KUKA KRL program: EPS_2_26115_SA7005_A_20260219035543.src

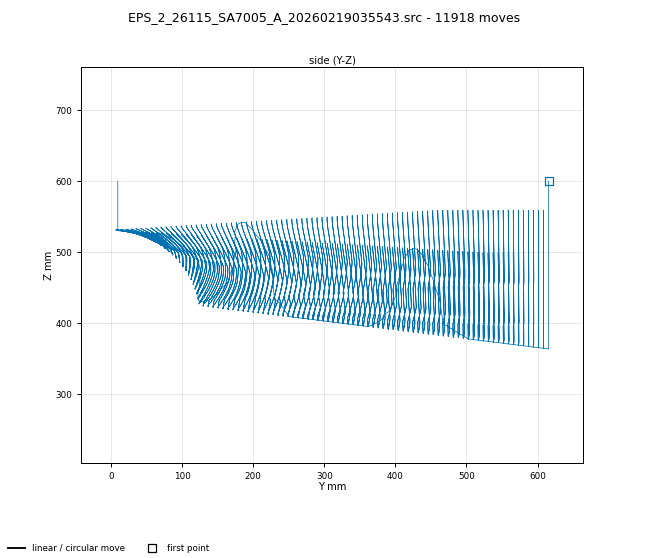
[picture p0: tool path of EPS_2_26115_SA7005_A_20260219035543.src, 11918 of 11920 moves have a stored position in this frame; points joined in program order, loops and branches not executed]
&ACCESS RVP
&REL 4
&COMMENT QRS 19112012
&PARAM EDITMASK = *
DEF PART()
EXT BAS (BAS_COMMAND :IN,REAL :IN )
INT I
BAS (#INITMOV,0 )

;KUKA QRS Post kuka4.cps  Date:22-06-2017 !

File_ID=3061

QRS_PRE_INIT()

;Init var - Until changes are made in qrs_pre_init
Outlet_Square_prg=0
Inlet_1_Square_prg=0
Inlet_2_Square_prg=0
Inlet_3_Square_prg=0
Inlet_4_Square_prg=0
Inlet_5_Square_prg=0

Outlet_1={X 0.000, Y 460.000, Z 458.500, B 0.000, E1 0.000 }
Inlet_1={X 0.000, Y 525.210, Z 398.500, B 0.000, E1 180.000 }
Outlet_1_type=201
Inlet_1_type=201
;QRS#1=Sidecore dimensions
;QRS#2=200-8" PVC SDR 35 Cut Back
;QRS#3=200-8" PVC SDR 35
;QRS#4=
;QRS#5=
;QRS#6=
;QRS#7=
;QRS#8=
;QRS#9=12-08 PSX
;QRS#10=12-08 PSX
;QRS#11=
;QRS#12=
;QRS#13=
;QRS#14=
;QRS#15=
;QRS#16=1220x127x838 2,75'
;QRS#17=EPS Height
;QRS#18=559
;QRS#19=*
;QRS#20= UPDATED VERSION 22-06-2017
;QRS#21=*
Outlet_Square=0100
Inlet_1_Square=0100
Inlet_2_Square=0
Inlet_3_Square=0
Inlet_4_Square=0
Inlet_5_Square=0
Mill_Square=1
Outlet_Square_Prg=214
Inlet_1_Square_prg=204

QRS_INIT()

$ADVANCE=5

; T1
PTP {E1 173.607,E2 173.607}
PTP {X 0,Y 615.507,A -85,B 0,C 180,E1 173.607,E2 173.607,E3 0,E4 0,E5 0,E6 0}
QRS_SPEED_INIT()
LIN {X 0,Y 615.507,Z 600,A -85,B 0,C 180,E1 173.607,E2 173.607,E3 0,E4 0,E5 0,E6 0} C_VEL
LIN {X 0,Y 615.507,Z 373.869,A -85,B 0,C 180,E1 173.607,E2 173.607} C_VEL
LIN {X 0,Y 615.507,Z 365.696,A -85,B 0,C 180,E1 173.607,E2 173.607} C_VEL
LIN {X 0,Y 615.492,Z 363.696,A -85,B 0,C 180,E1 173.421,E2 173.421} C_VEL
LIN {X 0,Y 615.49,Z 363.687,A -85,B 0,C 180,E1 170.801,E2 170.801} C_VEL
LIN {X 0,Y 615.487,Z 363.701,A -85,B 0,C 180,E1 168.139,E2 168.139} C_VEL
LIN {X 0,Y 615.481,Z 363.689,A -85,B 0,C 180,E1 165.451,E2 165.451} C_VEL
LIN {X 0,Y 615.493,Z 363.695,A -85,B 0,C 180,E1 162.73,E2 162.73} C_VEL
LIN {X 0,Y 615.49,Z 363.691,A -85,B 0,C 180,E1 159.967,E2 159.967} C_VEL
LIN {X 0,Y 615.483,Z 363.689,A -85,B 0,C 180,E1 157.155,E2 157.155} C_VEL
LIN {X 0,Y 615.486,Z 363.699,A -85,B 0,C 180,E1 154.284,E2 154.284} C_VEL
LIN {X 0,Y 615.478,Z 363.691,A -85,B 0,C 180,E1 151.552,E2 151.552} C_VEL
LIN {X 0,Y 615.487,Z 363.693,A -85,B 0,C 180,E1 148.915,E2 148.915} C_VEL
LIN {X 0,Y 615.478,Z 363.691,A -85,B 0,C 180,E1 146.468,E2 146.468} C_VEL
LIN {X 0,Y 615.493,Z 363.7,A -85,B 0,C 180,E1 144.166,E2 144.166} C_VEL
LIN {X 0,Y 615.483,Z 363.691,A -85,B 0,C 180,E1 141.931,E2 141.931} C_VEL
LIN {X 0,Y 615.482,Z 363.693,A -85,B 0,C 180,E1 139.393,E2 139.393} C_VEL
LIN {X 0,Y 615.478,Z 363.692,A -85,B 0,C 180,E1 136.754,E2 136.754} C_VEL
LIN {X 0,Y 615.491,Z 363.698,A -85,B 0,C 180,E1 133.997,E2 133.997} C_VEL
LIN {X 0,Y 615.49,Z 363.688,A -85,B 0,C 180,E1 131.474,E2 131.474} C_VEL
LIN {X 0,Y 615.49,Z 363.697,A -85,B 0,C 180,E1 128.904,E2 128.904} C_VEL
LIN {X 0,Y 615.485,Z 363.69,A -85,B 0,C 180,E1 126.425,E2 126.425} C_VEL
LIN {X 0,Y 615.485,Z 363.694,A -85,B 0,C 180,E1 125.616,E2 125.616} C_VEL
LIN {X 0,Y 615.494,Z 366.275,A -85,B 0,C 180,E1 123.236,E2 123.236} C_VEL
LIN {X 0,Y 615.479,Z 368.992,A -85,B 0,C 180,E1 120.92,E2 120.92} C_VEL
LIN {X 0,Y 615.491,Z 372.103,A -85,B 0,C 180,E1 118.45,E2 118.45} C_VEL
LIN {X 0,Y 615.498,Z 375.844,A -85,B 0,C 180,E1 115.57,E2 115.57} C_VEL
LIN {X 0,Y 615.489,Z 379.474,A -85,B 0,C 180,E1 112.845,E2 112.845} C_VEL
LIN {X 0,Y 615.479,Z 383.286,A -85,B 0,C 180,E1 110.033,E2 110.033} C_VEL
LIN {X 0,Y 615.493,Z 387.108,A -85,B 0,C 180,E1 107.27,E2 107.27} C_VEL
LIN {X 0,Y 615.482,Z 390.914,A -85,B 0,C 180,E1 104.549,E2 104.549} C_VEL
LIN {X 0,Y 615.495,Z 395.096,A -85,B 0,C 180,E1 101.61,E2 101.61} C_VEL
LIN {X 0,Y 615.494,Z 395.183,A -85,B 0,C 180,E1 101.548,E2 101.548} C_VEL
LIN {X 0,Y 615.481,Z 410.256,A -85,B 0,C 180,E1 101.193,E2 101.193} C_VEL
LIN {X 0,Y 615.494,Z 422.9,A -85,B 0,C 180,E1 100.751,E2 100.751} C_VEL
LIN {X 0,Y 615.479,Z 434.758,A -85,B 0,C 180,E1 100.195,E2 100.195} C_VEL
LIN {X 0,Y 615.499,Z 445.847,A -85,B 0,C 180,E1 99.53,E2 99.53} C_VEL
LIN {X 0,Y 615.498,Z 454.823,A -85,B 0,C 180,E1 98.867,E2 98.867} C_VEL
LIN {X 0,Y 615.498,Z 464.034,A -85,B 0,C 180,E1 98.041,E2 98.041} C_VEL
LIN {X 0,Y 615.499,Z 472.892,A -85,B 0,C 180,E1 97.057,E2 97.057} C_VEL
LIN {X 0,Y 615.497,Z 480.124,A -85,B 0,C 180,E1 96.063,E2 96.063} C_VEL
LIN {X 0,Y 615.497,Z 484.958,A -85,B 0,C 180,E1 95.241,E2 95.241} C_VEL
LIN {X 0,Y 615.494,Z 489.658,A -85,B 0,C 180,E1 94.256,E2 94.256} C_VEL
LIN {X 0,Y 615.494,Z 493.255,A -85,B 0,C 180,E1 93.273,E2 93.273} C_VEL
LIN {X 0,Y 615.496,Z 495.115,A -85,B 0,C 180,E1 92.618,E2 92.618} C_VEL
LIN {X 0,Y 615.5,Z 496.533,A -85,B 0,C 180,E1 91.963,E2 91.963} C_VEL
LIN {X 0,Y 615.496,Z 498.142,A -85,B 0,C 180,E1 90.654,E2 90.654} C_VEL
LIN {X 0,Y 615.495,Z 498.384,A -85,B 0,C 180,E1 90,E2 90} C_VEL
LIN {X 0,Y 615.495,Z 498.205,A -85,B 0,C 180,E1 89.346,E2 89.346} C_VEL
LIN {X 0,Y 615.5,Z 496.682,A -85,B 0,C 180,E1 88.037,E2 88.037} C_VEL
LIN {X 0,Y 615.498,Z 495.341,A -85,B 0,C 180,E1 87.382,E2 87.382} C_VEL
LIN {X 0,Y 615.496,Z 492.494,A -85,B 0,C 180,E1 86.399,E2 86.399} C_VEL
LIN {X 0,Y 615.498,Z 488.634,A -85,B 0,C 180,E1 85.415,E2 85.415} C_VEL
LIN {X 0,Y 615.498,Z 483.651,A -85,B 0,C 180,E1 84.43,E2 84.43} C_VEL
LIN {X 0,Y 615.496,Z 477.208,A -85,B 0,C 180,E1 83.418,E2 83.418} C_VEL
LIN {X 0,Y 615.497,Z 469.536,A -85,B 0,C 180,E1 82.454,E2 82.454} C_VEL
LIN {X 0,Y 615.498,Z 459.757,A -85,B 0,C 180,E1 81.463,E2 81.463} C_VEL
LIN {X 0,Y 615.498,Z 449.491,A -85,B 0,C 180,E1 80.636,E2 80.636} C_VEL
LIN {X 0,Y 615.482,Z 437.929,A -85,B 0,C 180,E1 79.888,E2 79.888} C_VEL
LIN {X 0,Y 615.491,Z 426.089,A -85,B 0,C 180,E1 79.294,E2 79.294} C_VEL
LIN {X 0,Y 615.477,Z 413.157,A -85,B 0,C 180,E1 78.807,E2 78.807} C_VEL
LIN {X 0,Y 615.486,Z 400.552,A -85,B 0,C 180,E1 78.473,E2 78.473} C_VEL
LIN {X 0,Y 615.494,Z 395.192,A -85,B 0,C 180,E1 78.369,E2 78.369} C_VEL
LIN {X 0,Y 615.482,Z 391.041,A -85,B 0,C 180,E1 75.451,E2 75.451} C_VEL
LIN {X 0,Y 615.497,Z 387.23,A -85,B 0,C 180,E1 72.73,E2 72.73} C_VEL
LIN {X 0,Y 615.479,Z 383.41,A -85,B 0,C 180,E1 69.967,E2 69.967} C_VEL
LIN {X 0,Y 615.492,Z 379.593,A -85,B 0,C 180,E1 67.155,E2 67.155} C_VEL
LIN {X 0,Y 615.487,Z 375.772,A -85,B 0,C 180,E1 64.284,E2 64.284} C_VEL
LIN {X 0,Y 615.492,Z 371.954,A -85,B 0,C 180,E1 61.342,E2 61.342} C_VEL
LIN {X 0,Y 615.483,Z 368.903,A -85,B 0,C 180,E1 58.915,E2 58.915} C_VEL
LIN {X 0,Y 615.495,Z 366.025,A -85,B 0,C 180,E1 56.465,E2 56.465} C_VEL
LIN {X 0,Y 615.484,Z 363.697,A -85,B 0,C 180,E1 54.384,E2 54.384} C_VEL
LIN {X 0,Y 615.481,Z 363.689,A -85,B 0,C 180,E1 51.931,E2 51.931} C_VEL
LIN {X 0,Y 615.494,Z 363.699,A -85,B 0,C 180,E1 49.394,E2 49.394} C_VEL
LIN {X 0,Y 615.496,Z 363.686,A -85,B 0,C 180,E1 46.756,E2 46.756} C_VEL
LIN {X 0,Y 615.486,Z 363.693,A -85,B 0,C 180,E1 43.997,E2 43.997} C_VEL
LIN {X 0,Y 615.488,Z 363.697,A -85,B 0,C 180,E1 41.094,E2 41.094} C_VEL
LIN {X 0,Y 615.495,Z 363.692,A -85,B 0,C 180,E1 38.904,E2 38.904} C_VEL
LIN {X 0,Y 615.478,Z 363.691,A -85,B 0,C 180,E1 36.426,E2 36.426} C_VEL
LIN {X 0,Y 615.495,Z 363.699,A -85,B 0,C 180,E1 34.022,E2 34.022} C_VEL
LIN {X 0,Y 615.482,Z 363.689,A -85,B 0,C 180,E1 31.686,E2 31.686} C_VEL
LIN {X 0,Y 615.478,Z 363.693,A -85,B 0,C 180,E1 29.407,E2 29.407} C_VEL
LIN {X 0,Y 615.498,Z 363.694,A -85,B 0,C 180,E1 27.046,E2 27.046} C_VEL
LIN {X 0,Y 615.487,Z 363.691,A -85,B 0,C 180,E1 24.272,E2 24.272} C_VEL
LIN {X 0,Y 615.479,Z 363.69,A -85,B 0,C 180,E1 21.432,E2 21.432} C_VEL
LIN {X 0,Y 615.486,Z 363.7,A -85,B 0,C 180,E1 18.603,E2 18.603} C_VEL
LIN {X 0,Y 615.477,Z 363.691,A -85,B 0,C 180,E1 15.906,E2 15.906} C_VEL
LIN {X 0,Y 615.494,Z 363.691,A -85,B 0,C 180,E1 13.201,E2 13.201} C_VEL
LIN {X 0,Y 615.486,Z 363.693,A -85,B 0,C 180,E1 10.527,E2 10.527} C_VEL
LIN {X 0,Y 615.477,Z 363.692,A -85,B 0,C 180,E1 7.876,E2 7.876} C_VEL
LIN {X 0,Y 615.496,Z 363.694,A -85,B 0,C 180,E1 5.241,E2 5.241} C_VEL
LIN {X 0,Y 615.488,Z 363.688,A -85,B 0,C 180,E1 2.618,E2 2.618} C_VEL
LIN {X 0,Y 615.487,Z 363.699,A -85,B 0,C 180,E1 0,E2 0} C_VEL
LIN {X 0,Y 615.488,Z 363.687,A -85,B 0,C 180,E1 -2.618,E2 -2.618} C_VEL
LIN {X 0,Y 615.494,Z 363.701,A -85,B 0,C 180,E1 -5.241,E2 -5.241} C_VEL
LIN {X 0,Y 615.478,Z 363.69,A -85,B 0,C 180,E1 -7.876,E2 -7.876} C_VEL
LIN {X 0,Y 615.486,Z 363.698,A -85,B 0,C 180,E1 -10.527,E2 -10.527} C_VEL
LIN {X 0,Y 615.494,Z 363.687,A -85,B 0,C 180,E1 -13.201,E2 -13.201} C_VEL
LIN {X 0,Y 615.487,Z 363.692,A -85,B 0,C 180,E1 -15.905,E2 -15.905} C_VEL
LIN {X 0,Y 615.488,Z 363.694,A -85,B 0,C 180,E1 -18.646,E2 -18.646} C_VEL
LIN {X 0,Y 615.478,Z 363.69,A -85,B 0,C 180,E1 -21.432,E2 -21.432} C_VEL
LIN {X 0,Y 615.484,Z 363.697,A -85,B 0,C 180,E1 -24.272,E2 -24.272} C_VEL
LIN {X 0,Y 615.497,Z 363.689,A -85,B 0,C 180,E1 -27.046,E2 -27.046} C_VEL
LIN {X 0,Y 615.488,Z 363.689,A -85,B 0,C 180,E1 -29.794,E2 -29.794} C_VEL
LIN {X 0,Y 615.491,Z 363.697,A -85,B 0,C 180,E1 -32.457,E2 -32.457} C_VEL
LIN {X 0,Y 615.49,Z 363.69,A -85,B 0,C 180,E1 -34.815,E2 -34.815} C_VEL
LIN {X 0,Y 615.481,Z 363.692,A -85,B 0,C 180,E1 -37.243,E2 -37.243} C_VEL
LIN {X 0,Y 615.483,Z 363.689,A -85,B 0,C 180,E1 -40.088,E2 -40.088} C_VEL
LIN {X 0,Y 615.477,Z 363.692,A -85,B 0,C 180,E1 -42.354,E2 -42.354} C_VEL
LIN {X 0,Y 615.48,Z 363.692,A -85,B 0,C 180,E1 -45.069,E2 -45.069} C_VEL
LIN {X 0,Y 615.495,Z 363.698,A -85,B 0,C 180,E1 -47.919,E2 -47.919} C_VEL
LIN {X 0,Y 615.477,Z 363.692,A -85,B 0,C 180,E1 -50.249,E2 -50.249} C_VEL
LIN {X 0,Y 615.483,Z 363.702,A -85,B 0,C 180,E1 -53.064,E2 -53.064} C_VEL
LIN {X 0,Y 615.49,Z 363.816,A -85,B 0,C 180,E1 -54.535,E2 -54.535} C_VEL
LIN {X 0,Y 615.482,Z 372.577,A -85,B 0,C 180,E1 -57.153,E2 -57.153} C_VEL
LIN {X 0,Y 615.484,Z 381.83,A -85,B 0,C 180,E1 -59.839,E2 -59.839} C_VEL
LIN {X 0,Y 615.495,Z 391.073,A -85,B 0,C 180,E1 -62.455,E2 -62.455} C_VEL
LIN {X 0,Y 615.478,Z 400.321,A -85,B 0,C 180,E1 -65.008,E2 -65.008} C_VEL
LIN {X 0,Y 615.479,Z 410.869,A -85,B 0,C 180,E1 -67.863,E2 -67.863} C_VEL
LIN {X 0,Y 615.48,Z 421.423,A -85,B 0,C 180,E1 -70.662,E2 -70.662} C_VEL
LIN {X 0,Y 615.489,Z 431.956,A -85,B 0,C 180,E1 -73.413,E2 -73.413} C_VEL
LIN {X 0,Y 615.492,Z 442.498,A -85,B 0,C 180,E1 -76.126,E2 -76.126} C_VEL
LIN {X 0,Y 615.491,Z 451.209,A -85,B 0,C 180,E1 -78.348,E2 -78.348} C_VEL
LIN {X 0,Y 615.499,Z 465.815,A -85,B 0,C 180,E1 -78.64,E2 -78.64} C_VEL
LIN {X 0,Y 615.489,Z 478.534,A -85,B 0,C 180,E1 -79.036,E2 -79.036} C_VEL
LIN {X 0,Y 615.479,Z 490.764,A -85,B 0,C 180,E1 -79.556,E2 -79.556} C_VEL
LIN {X 0,Y 615.498,Z 501.384,A -85,B 0,C 180,E1 -80.138,E2 -80.138} C_VEL
LIN {X 0,Y 615.498,Z 512.23,A -85,B 0,C 180,E1 -80.884,E2 -80.884} C_VEL
LIN {X 0,Y 615.497,Z 522.81,A -85,B 0,C 180,E1 -81.794,E2 -81.794} C_VEL
LIN {X 0,Y 615.498,Z 530.605,A -85,B 0,C 180,E1 -82.619,E2 -82.619} C_VEL
LIN {X 0,Y 615.496,Z 538.202,A -85,B 0,C 180,E1 -83.608,E2 -83.608} C_VEL
LIN {X 0,Y 615.498,Z 545.204,A -85,B 0,C 180,E1 -84.759,E2 -84.759} C_VEL
LIN {X 0,Y 615.493,Z 549.851,A -85,B 0,C 180,E1 -85.743,E2 -85.743} C_VEL
LIN {X 0,Y 615.495,Z 553.398,A -85,B 0,C 180,E1 -86.727,E2 -86.727} C_VEL
LIN {X 0,Y 615.497,Z 555.233,A -85,B 0,C 180,E1 -87.382,E2 -87.382} C_VEL
LIN {X 0,Y 615.499,Z 556.607,A -85,B 0,C 180,E1 -88.037,E2 -88.037} C_VEL
LIN {X 0,Y 615.496,Z 558.173,A -85,B 0,C 180,E1 -89.346,E2 -89.346} C_VEL
LIN {X 0,Y 615.494,Z 558.389,A -85,B 0,C 180,E1 -90,E2 -90} C_VEL
LIN {X 0,Y 615.496,Z 557.58,A -85,B 0,C 180,E1 -91.309,E2 -91.309} C_VEL
LIN {X 0,Y 615.499,Z 556.608,A -85,B 0,C 180,E1 -91.963,E2 -91.963} C_VEL
LIN {X 0,Y 615.497,Z 555.233,A -85,B 0,C 180,E1 -92.618,E2 -92.618} C_VEL
LIN {X 0,Y 615.496,Z 552.35,A -85,B 0,C 180,E1 -93.601,E2 -93.601} C_VEL
LIN {X 0,Y 615.498,Z 548.442,A -85,B 0,C 180,E1 -94.584,E2 -94.584} C_VEL
LIN {X 0,Y 615.499,Z 543.405,A -85,B 0,C 180,E1 -95.57,E2 -95.57} C_VEL
LIN {X 0,Y 615.497,Z 536.869,A -85,B 0,C 180,E1 -96.583,E2 -96.583} C_VEL
LIN {X 0,Y 615.497,Z 529.133,A -85,B 0,C 180,E1 -97.545,E2 -97.545} C_VEL
LIN {X 0,Y 615.498,Z 521.045,A -85,B 0,C 180,E1 -98.371,E2 -98.371} C_VEL
LIN {X 0,Y 615.499,Z 511.167,A -85,B 0,C 180,E1 -99.199,E2 -99.199} C_VEL
LIN {X 0,Y 615.491,Z 499.981,A -85,B 0,C 180,E1 -99.945,E2 -99.945} C_VEL
LIN {X 0,Y 615.481,Z 489.023,A -85,B 0,C 180,E1 -100.527,E2 -100.527} C_VEL
LIN {X 0,Y 615.489,Z 476.47,A -85,B 0,C 180,E1 -101.041,E2 -101.041} C_VEL
LIN {X 0,Y 615.498,Z 464.062,A -85,B 0,C 180,E1 -101.401,E2 -101.401} C_VEL
LIN {X 0,Y 615.491,Z 451.209,A -85,B 0,C 180,E1 -101.652,E2 -101.652} C_VEL
LIN {X 0,Y 615.476,Z 441.069,A -85,B 0,C 180,E1 -104.24,E2 -104.24} C_VEL
LIN {X 0,Y 615.484,Z 430.64,A -85,B 0,C 180,E1 -106.928,E2 -106.928} C_VEL
LIN {X 0,Y 615.485,Z 420.104,A -85,B 0,C 180,E1 -109.685,E2 -109.685} C_VEL
LIN {X 0,Y 615.492,Z 410.085,A -85,B 0,C 180,E1 -112.346,E2 -112.346} C_VEL
LIN {X 0,Y 615.481,Z 399.262,A -85,B 0,C 180,E1 -115.281,E2 -115.281} C_VEL
LIN {X 0,Y 615.487,Z 389.754,A -85,B 0,C 180,E1 -117.915,E2 -117.915} C_VEL
LIN {X 0,Y 615.496,Z 380.509,A -85,B 0,C 180,E1 -120.539,E2 -120.539} C_VEL
LIN {X 0,Y 615.491,Z 371.255,A -85,B 0,C 180,E1 -123.236,E2 -123.236} C_VEL
LIN {X 0,Y 615.489,Z 363.692,A -85,B 0,C 180,E1 -125.515,E2 -125.515} C_VEL
LIN {X 0,Y 615.481,Z 363.691,A -85,B 0,C 180,E1 -128.069,E2 -128.069} C_VEL
LIN {X 0,Y 615.482,Z 363.695,A -85,B 0,C 180,E1 -130.607,E2 -130.607} C_VEL
LIN {X 0,Y 615.496,Z 363.689,A -85,B 0,C 180,E1 -133.244,E2 -133.244} C_VEL
LIN {X 0,Y 615.488,Z 363.689,A -85,B 0,C 180,E1 -136.003,E2 -136.003} C_VEL
LIN {X 0,Y 615.489,Z 363.701,A -85,B 0,C 180,E1 -138.906,E2 -138.906} C_VEL
LIN {X 0,Y 615.49,Z 363.689,A -85,B 0,C 180,E1 -141.096,E2 -141.096} C_VEL
LIN {X 0,Y 615.478,Z 363.694,A -85,B 0,C 180,E1 -143.574,E2 -143.574} C_VEL
LIN {X 0,Y 615.494,Z 363.693,A -85,B 0,C 180,E1 -145.978,E2 -145.978} C_VEL
LIN {X 0,Y 615.482,Z 363.689,A -85,B 0,C 180,E1 -148.314,E2 -148.314} C_VEL
LIN {X 0,Y 615.481,Z 363.697,A -85,B 0,C 180,E1 -150.593,E2 -150.593} C_VEL
LIN {X 0,Y 615.497,Z 363.69,A -85,B 0,C 180,E1 -152.954,E2 -152.954} C_VEL
LIN {X 0,Y 615.484,Z 363.696,A -85,B 0,C 180,E1 -155.728,E2 -155.728} C_VEL
LIN {X 0,Y 615.478,Z 363.69,A -85,B 0,C 180,E1 -158.568,E2 -158.568} C_VEL
LIN {X 0,Y 615.489,Z 363.694,A -85,B 0,C 180,E1 -161.396,E2 -161.396} C_VEL
LIN {X 0,Y 615.486,Z 363.692,A -85,B 0,C 180,E1 -164.095,E2 -164.095} C_VEL
LIN {X 0,Y 615.494,Z 363.688,A -85,B 0,C 180,E1 -166.799,E2 -166.799} C_VEL
LIN {X 0,Y 615.486,Z 363.697,A -85,B 0,C 180,E1 -169.473,E2 -169.473} C_VEL
LIN {X 0,Y 615.478,Z 363.69,A -85,B 0,C 180,E1 -172.124,E2 -172.124} C_VEL
LIN {X 0,Y 615.491,Z 363.701,A -85,B 0,C 180,E1 -174.759,E2 -174.759} C_VEL
LIN {X 0,Y 615.488,Z 363.687,A -85,B 0,C 180,E1 -177.382,E2 -177.382} C_VEL
LIN {X 0,Y 615.486,Z 363.701,A -85,B 0,C 180,E1 -180,E2 -180} C_VEL
LIN {X 0,Y 615.488,Z 363.688,A -85,B 0,C 180,E1 -182.618,E2 -182.618} C_VEL
LIN {X 0,Y 615.495,Z 363.695,A -85,B 0,C 180,E1 -185.241,E2 -185.241} C_VEL
LIN {X 0,Y 615.492,Z 363.696,A -85,B 0,C 180,E1 -186.579,E2 -186.579} C_VEL
LIN {X 0,Y 614.816,Z 363.838,A -85,B 0,C 180,E1 -187.125,E2 -187.125} C_VEL
LIN {X 0,Y 611.982,Z 364.252,A -85,B 0,C 180,E1 -188.011,E2 -188.011} C_VEL
LIN {X 0,Y 609.59,Z 364.56,A -85,B 0,C 180,E1 -188.723,E2 -188.723} C_VEL
LIN {X 0,Y 608.552,Z 364.679,A -85,B 0,C 180,E1 -189.273,E2 -189.273} C_VEL
LIN {X 0,Y 608.462,Z 364.689,A -85,B 0,C 180,E1 -189.459,E2 -189.459} C_VEL
LIN {X 0,Y 608.463,Z 364.696,A -85,B 0,C 180,E1 -192,E2 -192} C_VEL
LIN {X 0,Y 608.473,Z 364.688,A -85,B 0,C 180,E1 -194.721,E2 -194.721} C_VEL
LIN {X 0,Y 608.455,Z 364.692,A -85,B 0,C 180,E1 -197.477,E2 -197.477} C_VEL
LIN {X 0,Y 608.469,Z 364.693,A -85,B 0,C 180,E1 -200.274,E2 -200.274} C_VEL
LIN {X 0,Y 608.449,Z 364.69,A -85,B 0,C 180,E1 -203.124,E2 -203.124} C_VEL
LIN {X 0,Y 608.475,Z 364.693,A -85,B 0,C 180,E1 -205.721,E2 -205.721} C_VEL
LIN {X 0,Y 608.446,Z 364.691,A -85,B 0,C 180,E1 -208.267,E2 -208.267} C_VEL
LIN {X 0,Y 608.476,Z 364.692,A -85,B 0,C 180,E1 -210.545,E2 -210.545} C_VEL
LIN {X 0,Y 608.459,Z 364.691,A -85,B 0,C 180,E1 -212.88,E2 -212.88} C_VEL
LIN {X 0,Y 608.443,Z 364.692,A -85,B 0,C 180,E1 -215.278,E2 -215.278} C_VEL
LIN {X 0,Y 608.469,Z 364.693,A -85,B 0,C 180,E1 -217.746,E2 -217.746} C_VEL
LIN {X 0,Y 608.448,Z 364.691,A -85,B 0,C 180,E1 -220.328,E2 -220.328} C_VEL
LIN {X 0,Y 608.449,Z 364.695,A -85,B 0,C 180,E1 -222.96,E2 -222.96} C_VEL
LIN {X 0,Y 608.461,Z 364.691,A -85,B 0,C 180,E1 -225.736,E2 -225.736} C_VEL
LIN {X 0,Y 608.465,Z 364.689,A -85,B 0,C 180,E1 -228.658,E2 -228.658} C_VEL
LIN {X 0,Y 608.465,Z 364.69,A -85,B 0,C 180,E1 -231.76,E2 -231.76} C_VEL
LIN {X 0,Y 608.447,Z 364.691,A -85,B 0,C 180,E1 -233.955,E2 -233.955} C_VEL
LIN {X 0,Y 608.413,Z 364.753,A -85,B 0,C 180,E1 -234.72,E2 -234.72} C_VEL
LIN {X 0,Y 608.433,Z 367.539,A -85,B 0,C 180,E1 -237.119,E2 -237.119} C_VEL
LIN {X 0,Y 608.426,Z 370.257,A -85,B 0,C 180,E1 -239.453,E2 -239.453} C_VEL
LIN {X 0,Y 608.433,Z 373.117,A -85,B 0,C 180,E1 -241.732,E2 -241.732} C_VEL
LIN {X 0,Y 608.438,Z 376.96,A -85,B 0,C 180,E1 -244.698,E2 -244.698} C_VEL
LIN {X 0,Y 608.436,Z 380.803,A -85,B 0,C 180,E1 -247.593,E2 -247.593} C_VEL
LIN {X 0,Y 608.414,Z 384.646,A -85,B 0,C 180,E1 -250.428,E2 -250.428} C_VEL
LIN {X 0,Y 608.42,Z 388.49,A -85,B 0,C 180,E1 -253.215,E2 -253.215} C_VEL
LIN {X 0,Y 608.442,Z 392.379,A -85,B 0,C 180,E1 -255.994,E2 -255.994} C_VEL
LIN {X 0,Y 608.444,Z 395.666,A -85,B 0,C 180,E1 -258.317,E2 -258.317} C_VEL
LIN {X 0,Y 608.531,Z 411.501,A -85,B 0,C 180,E1 -258.71,E2 -258.71} C_VEL
LIN {X 0,Y 608.516,Z 423.818,A -85,B 0,C 180,E1 -259.157,E2 -259.157} C_VEL
LIN {X 0,Y 608.48,Z 434.934,A -85,B 0,C 180,E1 -259.687,E2 -259.687} C_VEL
LIN {X 0,Y 608.5,Z 446.067,A -85,B 0,C 180,E1 -260.359,E2 -260.359} C_VEL
LIN {X 0,Y 608.474,Z 455.084,A -85,B 0,C 180,E1 -261.029,E2 -261.029} C_VEL
LIN {X 0,Y 608.464,Z 464.35,A -85,B 0,C 180,E1 -261.866,E2 -261.866} C_VEL
LIN {X 0,Y 608.466,Z 473.323,A -85,B 0,C 180,E1 -262.867,E2 -262.867} C_VEL
LIN {X 0,Y 608.444,Z 480.555,A -85,B 0,C 180,E1 -263.867,E2 -263.867} C_VEL
LIN {X 0,Y 608.462,Z 485.434,A -85,B 0,C 180,E1 -264.698,E2 -264.698} C_VEL
LIN {X 0,Y 608.439,Z 490.178,A -85,B 0,C 180,E1 -265.694,E2 -265.694} C_VEL
LIN {X 0,Y 608.425,Z 493.812,A -85,B 0,C 180,E1 -266.689,E2 -266.689} C_VEL
LIN {X 0,Y 608.425,Z 495.691,A -85,B 0,C 180,E1 -267.352,E2 -267.352} C_VEL
LIN {X 0,Y 608.444,Z 497.127,A -85,B 0,C 180,E1 -268.014,E2 -268.014} C_VEL
LIN {X 0,Y 608.439,Z 498.752,A -85,B 0,C 180,E1 -269.338,E2 -269.338} C_VEL
LIN {X 0,Y 608.435,Z 498.995,A -85,B 0,C 180,E1 -270,E2 -270} C_VEL
LIN {X 0,Y 608.438,Z 498.815,A -85,B 0,C 180,E1 -270.662,E2 -270.662} C_VEL
LIN {X 0,Y 608.445,Z 497.276,A -85,B 0,C 180,E1 -271.986,E2 -271.986} C_VEL
LIN {X 0,Y 608.426,Z 495.918,A -85,B 0,C 180,E1 -272.648,E2 -272.648} C_VEL
LIN {X 0,Y 608.449,Z 493.041,A -85,B 0,C 180,E1 -273.642,E2 -273.642} C_VEL
LIN {X 0,Y 608.433,Z 489.142,A -85,B 0,C 180,E1 -274.638,E2 -274.638} C_VEL
LIN {X 0,Y 608.45,Z 484.111,A -85,B 0,C 180,E1 -275.635,E2 -275.635} C_VEL
LIN {X 0,Y 608.441,Z 477.794,A -85,B 0,C 180,E1 -276.633,E2 -276.633} C_VEL
LIN {X 0,Y 608.475,Z 469.877,A -85,B 0,C 180,E1 -277.633,E2 -277.633} C_VEL
LIN {X 0,Y 608.472,Z 460.035,A -85,B 0,C 180,E1 -278.636,E2 -278.636} C_VEL
LIN {X 0,Y 608.481,Z 449.712,A -85,B 0,C 180,E1 -279.473,E2 -279.473} C_VEL
LIN {X 0,Y 608.478,Z 438.097,A -85,B 0,C 180,E1 -280.229,E2 -280.229} C_VEL
LIN {X 0,Y 608.507,Z 426.22,A -85,B 0,C 180,E1 -280.831,E2 -280.831} C_VEL
LIN {X 0,Y 608.521,Z 413.257,A -85,B 0,C 180,E1 -281.323,E2 -281.323} C_VEL
LIN {X 0,Y 608.546,Z 400.638,A -85,B 0,C 180,E1 -281.66,E2 -281.66} C_VEL
LIN {X 0,Y 608.441,Z 395.674,A -85,B 0,C 180,E1 -281.768,E2 -281.768} C_VEL
LIN {X 0,Y 608.423,Z 392.46,A -85,B 0,C 180,E1 -284.039,E2 -284.039} C_VEL
LIN {X 0,Y 608.421,Z 388.615,A -85,B 0,C 180,E1 -286.785,E2 -286.785} C_VEL
LIN {X 0,Y 608.416,Z 384.769,A -85,B 0,C 180,E1 -289.572,E2 -289.572} C_VEL
LIN {X 0,Y 608.433,Z 380.84,A -85,B 0,C 180,E1 -292.469,E2 -292.469} C_VEL
LIN {X 0,Y 608.438,Z 377.078,A -85,B 0,C 180,E1 -295.302,E2 -295.302} C_VEL
LIN {X 0,Y 608.433,Z 373.232,A -85,B 0,C 180,E1 -298.268,E2 -298.268} C_VEL
LIN {X 0,Y 608.429,Z 370.361,A -85,B 0,C 180,E1 -300.547,E2 -300.547} C_VEL
LIN {X 0,Y 608.434,Z 367.65,A -85,B 0,C 180,E1 -302.881,E2 -302.881} C_VEL
LIN {X 0,Y 608.44,Z 364.856,A -85,B 0,C 180,E1 -305.278,E2 -305.278} C_VEL
LIN {X 0,Y 608.469,Z 364.689,A -85,B 0,C 180,E1 -307.747,E2 -307.747} C_VEL
LIN {X 0,Y 608.453,Z 364.695,A -85,B 0,C 180,E1 -310.329,E2 -310.329} C_VEL
LIN {X 0,Y 608.483,Z 364.687,A -85,B 0,C 180,E1 -313.31,E2 -313.31} C_VEL
LIN {X 0,Y 608.47,Z 364.69,A -85,B 0,C 180,E1 -316.13,E2 -316.13} C_VEL
LIN {X 0,Y 608.456,Z 364.694,A -85,B 0,C 180,E1 -318.823,E2 -318.823} C_VEL
LIN {X 0,Y 608.474,Z 364.688,A -85,B 0,C 180,E1 -321.412,E2 -321.412} C_VEL
LIN {X 0,Y 608.453,Z 364.694,A -85,B 0,C 180,E1 -323.954,E2 -323.954} C_VEL
LIN {X 0,Y 608.45,Z 364.693,A -85,B 0,C 180,E1 -326.328,E2 -326.328} C_VEL
LIN {X 0,Y 608.45,Z 364.691,A -85,B 0,C 180,E1 -328.733,E2 -328.733} C_VEL
LIN {X 0,Y 608.468,Z 364.691,A -85,B 0,C 180,E1 -331.382,E2 -331.382} C_VEL
LIN {X 0,Y 608.438,Z 364.693,A -85,B 0,C 180,E1 -333.964,E2 -333.964} C_VEL
LIN {X 0,Y 608.473,Z 364.696,A -85,B 0,C 180,E1 -336.155,E2 -336.155} C_VEL
LIN {X 0,Y 608.456,Z 364.69,A -85,B 0,C 180,E1 -339.018,E2 -339.018} C_VEL
LIN {X 0,Y 608.447,Z 364.692,A -85,B 0,C 180,E1 -341.828,E2 -341.828} C_VEL
LIN {X 0,Y 608.471,Z 364.694,A -85,B 0,C 180,E1 -344.594,E2 -344.594} C_VEL
LIN {X 0,Y 608.476,Z 364.687,A -85,B 0,C 180,E1 -347.323,E2 -347.323} C_VEL
LIN {X 0,Y 608.456,Z 364.695,A -85,B 0,C 180,E1 -350.023,E2 -350.023} C_VEL
LIN {X 0,Y 608.466,Z 364.689,A -85,B 0,C 180,E1 -352.701,E2 -352.701} C_VEL
LIN {X 0,Y 608.457,Z 364.692,A -85,B 0,C 180,E1 -355.362,E2 -355.362} C_VEL
LIN {X 0,Y 608.45,Z 364.693,A -85,B 0,C 180,E1 -358.014,E2 -358.014} C_VEL
LIN {X 0,Y 608.479,Z 364.688,A -85,B 0,C 180,E1 -360.662,E2 -360.662} C_VEL
LIN {X 0,Y 608.478,Z 364.691,A -85,B 0,C 180,E1 -363.311,E2 -363.311} C_VEL
LIN {X 0,Y 608.454,Z 364.69,A -85,B 0,C 180,E1 -365.967,E2 -365.967} C_VEL
LIN {X 0,Y 608.465,Z 364.696,A -85,B 0,C 180,E1 -368.636,E2 -368.636} C_VEL
LIN {X 0,Y 608.478,Z 364.687,A -85,B 0,C 180,E1 -371.324,E2 -371.324} C_VEL
LIN {X 0,Y 608.476,Z 364.692,A -85,B 0,C 180,E1 -374.037,E2 -374.037} C_VEL
LIN {X 0,Y 608.445,Z 364.693,A -85,B 0,C 180,E1 -376.784,E2 -376.784} C_VEL
LIN {X 0,Y 608.455,Z 364.69,A -85,B 0,C 180,E1 -379.571,E2 -379.571} C_VEL
LIN {X 0,Y 608.464,Z 364.695,A -85,B 0,C 180,E1 -382.476,E2 -382.476} C_VEL
LIN {X 0,Y 608.456,Z 364.691,A -85,B 0,C 180,E1 -384.571,E2 -384.571} C_VEL
LIN {X 0,Y 608.487,Z 364.69,A -85,B 0,C 180,E1 -387.208,E2 -387.208} C_VEL
LIN {X 0,Y 608.47,Z 364.688,A -85,B 0,C 180,E1 -389.971,E2 -389.971} C_VEL
LIN {X 0,Y 608.458,Z 364.693,A -85,B 0,C 180,E1 -392.88,E2 -392.88} C_VEL
LIN {X 0,Y 608.442,Z 364.692,A -85,B 0,C 180,E1 -395.278,E2 -395.278} C_VEL
LIN {X 0,Y 608.467,Z 364.696,A -85,B 0,C 180,E1 -397.747,E2 -397.747} C_VEL
LIN {X 0,Y 608.447,Z 364.691,A -85,B 0,C 180,E1 -400.328,E2 -400.328} C_VEL
LIN {X 0,Y 608.454,Z 364.697,A -85,B 0,C 180,E1 -402.96,E2 -402.96} C_VEL
LIN {X 0,Y 608.463,Z 364.69,A -85,B 0,C 180,E1 -405.736,E2 -405.736} C_VEL
LIN {X 0,Y 608.464,Z 364.689,A -85,B 0,C 180,E1 -408.658,E2 -408.658} C_VEL
LIN {X 0,Y 608.464,Z 364.692,A -85,B 0,C 180,E1 -411.76,E2 -411.76} C_VEL
LIN {X 0,Y 608.482,Z 364.814,A -85,B 0,C 180,E1 -414.369,E2 -414.369} C_VEL
LIN {X 0,Y 608.528,Z 372.592,A -85,B 0,C 180,E1 -416.73,E2 -416.73} C_VEL
LIN {X 0,Y 608.536,Z 381.859,A -85,B 0,C 180,E1 -419.459,E2 -419.459} C_VEL
LIN {X 0,Y 608.509,Z 392.45,A -85,B 0,C 180,E1 -422.485,E2 -422.485} C_VEL
LIN {X 0,Y 608.469,Z 401.718,A -85,B 0,C 180,E1 -425.065,E2 -425.065} C_VEL
LIN {X 0,Y 608.479,Z 412.309,A -85,B 0,C 180,E1 -427.952,E2 -427.952} C_VEL
LIN {X 0,Y 608.453,Z 422.9,A -85,B 0,C 180,E1 -430.78,E2 -430.78} C_VEL
LIN {X 0,Y 608.442,Z 433.181,A -85,B 0,C 180,E1 -433.48,E2 -433.48} C_VEL
LIN {X 0,Y 608.446,Z 444.146,A -85,B 0,C 180,E1 -436.319,E2 -436.319} C_VEL
LIN {X 0,Y 608.442,Z 451.53,A -85,B 0,C 180,E1 -438.211,E2 -438.211} C_VEL
LIN {X 0,Y 608.544,Z 466.691,A -85,B 0,C 180,E1 -438.53,E2 -438.53} C_VEL
LIN {X 0,Y 608.526,Z 478.239,A -85,B 0,C 180,E1 -438.893,E2 -438.893} C_VEL
LIN {X 0,Y 608.51,Z 490.918,A -85,B 0,C 180,E1 -439.435,E2 -439.435} C_VEL
LIN {X 0,Y 608.489,Z 501.576,A -85,B 0,C 180,E1 -440.023,E2 -440.023} C_VEL
LIN {X 0,Y 608.483,Z 512.472,A -85,B 0,C 180,E1 -440.778,E2 -440.778} C_VEL
LIN {X 0,Y 608.475,Z 523.11,A -85,B 0,C 180,E1 -441.699,E2 -441.699} C_VEL
LIN {X 0,Y 608.471,Z 530.959,A -85,B 0,C 180,E1 -442.534,E2 -442.534} C_VEL
LIN {X 0,Y 608.461,Z 538.286,A -85,B 0,C 180,E1 -443.484,E2 -443.484} C_VEL
LIN {X 0,Y 608.45,Z 543.865,A -85,B 0,C 180,E1 -444.365,E2 -444.365} C_VEL
LIN {X 0,Y 608.432,Z 548.95,A -85,B 0,C 180,E1 -445.362,E2 -445.362} C_VEL
LIN {X 0,Y 608.449,Z 552.896,A -85,B 0,C 180,E1 -446.358,E2 -446.358} C_VEL
LIN {X 0,Y 608.425,Z 555.809,A -85,B 0,C 180,E1 -447.352,E2 -447.352} C_VEL
LIN {X 0,Y 608.444,Z 557.201,A -85,B 0,C 180,E1 -448.014,E2 -448.014} C_VEL
LIN {X 0,Y 608.438,Z 558.783,A -85,B 0,C 180,E1 -449.338,E2 -449.338} C_VEL
LIN {X 0,Y 608.434,Z 559,A -85,B 0,C 180,E1 -450,E2 -450} C_VEL
LIN {X 0,Y 608.448,Z 558.184,A -85,B 0,C 180,E1 -451.324,E2 -451.324} C_VEL
LIN {X 0,Y 608.444,Z 557.201,A -85,B 0,C 180,E1 -451.986,E2 -451.986} C_VEL
LIN {X 0,Y 608.425,Z 555.809,A -85,B 0,C 180,E1 -452.648,E2 -452.648} C_VEL
LIN {X 0,Y 608.449,Z 552.896,A -85,B 0,C 180,E1 -453.642,E2 -453.642} C_VEL
LIN {X 0,Y 608.432,Z 548.95,A -85,B 0,C 180,E1 -454.638,E2 -454.638} C_VEL
LIN {X 0,Y 608.437,Z 542.877,A -85,B 0,C 180,E1 -455.801,E2 -455.801} C_VEL
LIN {X 0,Y 608.462,Z 536.235,A -85,B 0,C 180,E1 -456.799,E2 -456.799} C_VEL
LIN {X 0,Y 608.456,Z 527.989,A -85,B 0,C 180,E1 -457.8,E2 -457.8} C_VEL
LIN {X 0,Y 608.472,Z 519.536,A -85,B 0,C 180,E1 -458.636,E2 -458.636} C_VEL
LIN {X 0,Y 608.481,Z 509.09,A -85,B 0,C 180,E1 -459.473,E2 -459.473} C_VEL
LIN {X 0,Y 608.491,Z 498.755,A -85,B 0,C 180,E1 -460.145,E2 -460.145} C_VEL
LIN {X 0,Y 608.518,Z 487.259,A -85,B 0,C 180,E1 -460.74,E2 -460.74} C_VEL
LIN {X 0,Y 608.537,Z 474.891,A -85,B 0,C 180,E1 -461.225,E2 -461.225} C_VEL
LIN {X 0,Y 608.546,Z 461.438,A -85,B 0,C 180,E1 -461.597,E2 -461.597} C_VEL
LIN {X 0,Y 608.442,Z 451.53,A -85,B 0,C 180,E1 -461.789,E2 -461.789} C_VEL
LIN {X 0,Y 608.442,Z 441.435,A -85,B 0,C 180,E1 -464.379,E2 -464.379} C_VEL
LIN {X 0,Y 608.442,Z 430.844,A -85,B 0,C 180,E1 -467.13,E2 -467.13} C_VEL
LIN {X 0,Y 608.458,Z 421.577,A -85,B 0,C 180,E1 -469.57,E2 -469.57} C_VEL
LIN {X 0,Y 608.467,Z 410.72,A -85,B 0,C 180,E1 -472.477,E2 -472.477} C_VEL
LIN {X 0,Y 608.473,Z 400.394,A -85,B 0,C 180,E1 -475.3,E2 -475.3} C_VEL
LIN {X 0,Y 608.5,Z 391.127,A -85,B 0,C 180,E1 -477.889,E2 -477.889} C_VEL
LIN {X 0,Y 608.536,Z 381.859,A -85,B 0,C 180,E1 -480.541,E2 -480.541} C_VEL
LIN {X 0,Y 608.528,Z 372.592,A -85,B 0,C 180,E1 -483.27,E2 -483.27} C_VEL
LIN {X 0,Y 608.475,Z 364.691,A -85,B 0,C 180,E1 -485.682,E2 -485.682} C_VEL
LIN {X 0,Y 608.464,Z 364.692,A -85,B 0,C 180,E1 -488.24,E2 -488.24} C_VEL
LIN {X 0,Y 608.463,Z 364.689,A -85,B 0,C 180,E1 -491.342,E2 -491.342} C_VEL
LIN {X 0,Y 608.463,Z 364.69,A -85,B 0,C 180,E1 -494.264,E2 -494.264} C_VEL
LIN {X 0,Y 608.45,Z 364.697,A -85,B 0,C 180,E1 -497.04,E2 -497.04} C_VEL
LIN {X 0,Y 608.456,Z 364.69,A -85,B 0,C 180,E1 -499.697,E2 -499.697} C_VEL
LIN {X 0,Y 608.467,Z 364.696,A -85,B 0,C 180,E1 -502.253,E2 -502.253} C_VEL
LIN {X 0,Y 608.454,Z 364.691,A -85,B 0,C 180,E1 -505.094,E2 -505.094} C_VEL
LIN {X 0,Y 608.468,Z 364.69,A -85,B 0,C 180,E1 -507.906,E2 -507.906} C_VEL
LIN {X 0,Y 608.473,Z 364.688,A -85,B 0,C 180,E1 -510.221,E2 -510.221} C_VEL
LIN {X 0,Y 608.487,Z 364.69,A -85,B 0,C 180,E1 -512.792,E2 -512.792} C_VEL
LIN {X 0,Y 608.455,Z 364.691,A -85,B 0,C 180,E1 -515.429,E2 -515.429} C_VEL
LIN {X 0,Y 608.468,Z 364.689,A -85,B 0,C 180,E1 -518.308,E2 -518.308} C_VEL
LIN {X 0,Y 608.46,Z 364.697,A -85,B 0,C 180,E1 -521.13,E2 -521.13} C_VEL
LIN {X 0,Y 608.461,Z 364.69,A -85,B 0,C 180,E1 -523.906,E2 -523.906} C_VEL
LIN {X 0,Y 608.472,Z 364.69,A -85,B 0,C 180,E1 -526.644,E2 -526.644} C_VEL
LIN {X 0,Y 608.462,Z 364.692,A -85,B 0,C 180,E1 -529.35,E2 -529.35} C_VEL
LIN {X 0,Y 608.474,Z 364.688,A -85,B 0,C 180,E1 -532.033,E2 -532.033} C_VEL
LIN {X 0,Y 608.469,Z 364.695,A -85,B 0,C 180,E1 -534.698,E2 -534.698} C_VEL
LIN {X 0,Y 608.479,Z 364.687,A -85,B 0,C 180,E1 -537.352,E2 -537.352} C_VEL
LIN {X 0,Y 608.478,Z 364.694,A -85,B 0,C 180,E1 -540,E2 -540} C_VEL
LIN {X 0,Y 608.479,Z 364.687,A -85,B 0,C 180,E1 -542.648,E2 -542.648} C_VEL
LIN {X 0,Y 608.473,Z 364.692,A -85,B 0,C 180,E1 -545.302,E2 -545.302} C_VEL
LIN {X 0,Y 608.473,Z 364.689,A -85,B 0,C 180,E1 -547.967,E2 -547.967} C_VEL
LIN {X 0,Y 608.462,Z 364.689,A -85,B 0,C 180,E1 -549.459,E2 -549.459} C_VEL
LIN {X 0,Y 607.78,Z 364.781,A -85,B 0,C 180,E1 -550.012,E2 -550.012} C_VEL
LIN {X 0,Y 604.925,Z 365.135,A -85,B 0,C 180,E1 -550.908,E2 -550.908} C_VEL
LIN {X 0,Y 602.524,Z 365.435,A -85,B 0,C 180,E1 -551.63,E2 -551.63} C_VEL
LIN {X 0,Y 601.494,Z 365.561,A -85,B 0,C 180,E1 -552.187,E2 -552.187} C_VEL
LIN {X 0,Y 601.411,Z 365.569,A -85,B 0,C 180,E1 -552.375,E2 -552.375} C_VEL
LIN {X 0,Y 601.429,Z 365.567,A -85,B 0,C 180,E1 -554.897,E2 -554.897} C_VEL
LIN {X 0,Y 601.426,Z 365.573,A -85,B 0,C 180,E1 -556.986,E2 -556.986} C_VEL
LIN {X 0,Y 601.411,Z 365.568,A -85,B 0,C 180,E1 -559.809,E2 -559.809} C_VEL
LIN {X 0,Y 601.416,Z 365.568,A -85,B 0,C 180,E1 -562.683,E2 -562.683} C_VEL
LIN {X 0,Y 601.408,Z 365.568,A -85,B 0,C 180,E1 -564.878,E2 -564.878} C_VEL
LIN {X 0,Y 601.423,Z 365.573,A -85,B 0,C 180,E1 -567.363,E2 -567.363} C_VEL
LIN {X 0,Y 601.433,Z 365.566,A -85,B 0,C 180,E1 -570.164,E2 -570.164} C_VEL
LIN {X 0,Y 601.427,Z 365.569,A -85,B 0,C 180,E1 -572.716,E2 -572.716} C_VEL
LIN {X 0,Y 601.401,Z 365.569,A -85,B 0,C 180,E1 -575.112,E2 -575.112} C_VEL
LIN {X 0,Y 601.439,Z 365.569,A -85,B 0,C 180,E1 -577.419,E2 -577.419} C_VEL
LIN {X 0,Y 601.415,Z 365.567,A -85,B 0,C 180,E1 -579.995,E2 -579.995} C_VEL
LIN {X 0,Y 601.41,Z 365.575,A -85,B 0,C 180,E1 -582.671,E2 -582.671} C_VEL
LIN {X 0,Y 601.43,Z 365.565,A -85,B 0,C 180,E1 -585.482,E2 -585.482} C_VEL
LIN {X 0,Y 601.429,Z 365.566,A -85,B 0,C 180,E1 -588.407,E2 -588.407} C_VEL
LIN {X 0,Y 601.435,Z 365.569,A -85,B 0,C 180,E1 -591.529,E2 -591.529} C_VEL
LIN {X 0,Y 601.379,Z 365.573,A -85,B 0,C 180,E1 -594.245,E2 -594.245} C_VEL
LIN {X 0,Y 601.357,Z 365.822,A -85,B 0,C 180,E1 -595.064,E2 -595.064} C_VEL
LIN {X 0,Y 601.378,Z 368.588,A -85,B 0,C 180,E1 -597.481,E2 -597.481} C_VEL
LIN {X 0,Y 601.355,Z 371.32,A -85,B 0,C 180,E1 -599.864,E2 -599.864} C_VEL
LIN {X 0,Y 601.345,Z 374.743,A -85,B 0,C 180,E1 -602.651,E2 -602.651} C_VEL
LIN {X 0,Y 601.349,Z 377.922,A -85,B 0,C 180,E1 -605.119,E2 -605.119} C_VEL
LIN {X 0,Y 601.337,Z 381.765,A -85,B 0,C 180,E1 -608.038,E2 -608.038} C_VEL
LIN {X 0,Y 601.316,Z 384.647,A -85,B 0,C 180,E1 -610.187,E2 -610.187} C_VEL
LIN {X 0,Y 601.338,Z 388.49,A -85,B 0,C 180,E1 -613.011,E2 -613.011} C_VEL
LIN {X 0,Y 601.35,Z 392.534,A -85,B 0,C 180,E1 -615.937,E2 -615.937} C_VEL
LIN {X 0,Y 601.347,Z 395.667,A -85,B 0,C 180,E1 -618.177,E2 -618.177} C_VEL
LIN {X 0,Y 601.591,Z 401.34,A -85,B 0,C 180,E1 -618.31,E2 -618.31} C_VEL
LIN {X 0,Y 601.557,Z 414.026,A -85,B 0,C 180,E1 -618.66,E2 -618.66} C_VEL
LIN {X 0,Y 601.543,Z 426.615,A -85,B 0,C 180,E1 -619.15,E2 -619.15} C_VEL
LIN {X 0,Y 601.503,Z 438.007,A -85,B 0,C 180,E1 -619.736,E2 -619.736} C_VEL
LIN {X 0,Y 601.462,Z 449.637,A -85,B 0,C 180,E1 -620.5,E2 -620.5} C_VEL
LIN {X 0,Y 601.436,Z 459.023,A -85,B 0,C 180,E1 -621.262,E2 -621.262} C_VEL
LIN {X 0,Y 601.4,Z 467.59,A -85,B 0,C 180,E1 -622.108,E2 -622.108} C_VEL
LIN {X 0,Y 601.388,Z 475.906,A -85,B 0,C 180,E1 -623.12,E2 -623.12} C_VEL
LIN {X 0,Y 601.373,Z 482.607,A -85,B 0,C 180,E1 -624.131,E2 -624.131} C_VEL
LIN {X 0,Y 601.335,Z 488.754,A -85,B 0,C 180,E1 -625.307,E2 -625.307} C_VEL
LIN {X 0,Y 601.367,Z 492.743,A -85,B 0,C 180,E1 -626.315,E2 -626.315} C_VEL
LIN {X 0,Y 601.324,Z 495.693,A -85,B 0,C 180,E1 -627.32,E2 -627.32} C_VEL
LIN {X 0,Y 601.343,Z 497.127,A -85,B 0,C 180,E1 -627.991,E2 -627.991} C_VEL
LIN {X 0,Y 601.339,Z 498.753,A -85,B 0,C 180,E1 -629.33,E2 -629.33} C_VEL
LIN {X 0,Y 601.336,Z 498.996,A -85,B 0,C 180,E1 -630,E2 -630} C_VEL
LIN {X 0,Y 601.339,Z 498.815,A -85,B 0,C 180,E1 -630.67,E2 -630.67} C_VEL
LIN {X 0,Y 601.343,Z 497.275,A -85,B 0,C 180,E1 -632.009,E2 -632.009} C_VEL
LIN {X 0,Y 601.326,Z 495.916,A -85,B 0,C 180,E1 -632.68,E2 -632.68} C_VEL
LIN {X 0,Y 601.368,Z 493.04,A -85,B 0,C 180,E1 -633.685,E2 -633.685} C_VEL
LIN {X 0,Y 601.337,Z 489.14,A -85,B 0,C 180,E1 -634.693,E2 -634.693} C_VEL
LIN {X 0,Y 601.373,Z 484.109,A -85,B 0,C 180,E1 -635.701,E2 -635.701} C_VEL
LIN {X 0,Y 601.382,Z 477.79,A -85,B 0,C 180,E1 -636.711,E2 -636.711} C_VEL
LIN {X 0,Y 601.396,Z 469.873,A -85,B 0,C 180,E1 -637.724,E2 -637.724} C_VEL
LIN {X 0,Y 601.437,Z 460.028,A -85,B 0,C 180,E1 -638.738,E2 -638.738} C_VEL
LIN {X 0,Y 601.451,Z 449.706,A -85,B 0,C 180,E1 -639.585,E2 -639.585} C_VEL
LIN {X 0,Y 601.481,Z 438.087,A -85,B 0,C 180,E1 -640.349,E2 -640.349} C_VEL
LIN {X 0,Y 601.523,Z 426.209,A -85,B 0,C 180,E1 -640.958,E2 -640.958} C_VEL
LIN {X 0,Y 601.543,Z 413.241,A -85,B 0,C 180,E1 -641.456,E2 -641.456} C_VEL
LIN {X 0,Y 601.614,Z 400.615,A -85,B 0,C 180,E1 -641.796,E2 -641.796} C_VEL
LIN {X 0,Y 601.342,Z 395.673,A -85,B 0,C 180,E1 -641.909,E2 -641.909} C_VEL
LIN {X 0,Y 601.319,Z 392.459,A -85,B 0,C 180,E1 -644.208,E2 -644.208} C_VEL
LIN {X 0,Y 601.34,Z 388.614,A -85,B 0,C 180,E1 -646.989,E2 -646.989} C_VEL
LIN {X 0,Y 601.317,Z 384.768,A -85,B 0,C 180,E1 -649.813,E2 -649.813} C_VEL
LIN {X 0,Y 601.337,Z 381.055,A -85,B 0,C 180,E1 -652.587,E2 -652.587} C_VEL
LIN {X 0,Y 601.349,Z 378.039,A -85,B 0,C 180,E1 -654.881,E2 -654.881} C_VEL
LIN {X 0,Y 601.346,Z 374.858,A -85,B 0,C 180,E1 -657.349,E2 -657.349} C_VEL
LIN {X 0,Y 601.352,Z 371.368,A -85,B 0,C 180,E1 -660.169,E2 -660.169} C_VEL
LIN {X 0,Y 601.366,Z 368.513,A -85,B 0,C 180,E1 -662.707,E2 -662.707} C_VEL
LIN {X 0,Y 601.384,Z 365.723,A -85,B 0,C 180,E1 -665.11,E2 -665.11} C_VEL
LIN {X 0,Y 601.44,Z 365.567,A -85,B 0,C 180,E1 -667.419,E2 -667.419} C_VEL
LIN {X 0,Y 601.406,Z 365.569,A -85,B 0,C 180,E1 -669.996,E2 -669.996} C_VEL
LIN {X 0,Y 601.416,Z 365.569,A -85,B 0,C 180,E1 -672.67,E2 -672.67} C_VEL
LIN {X 0,Y 601.43,Z 365.566,A -85,B 0,C 180,E1 -674.535,E2 -674.535} C_VEL
LIN {X 0,Y 601.411,Z 365.575,A -85,B 0,C 180,E1 -677.41,E2 -677.41} C_VEL
LIN {X 0,Y 601.446,Z 365.566,A -85,B 0,C 180,E1 -680.464,E2 -680.464} C_VEL
LIN {X 0,Y 601.407,Z 365.568,A -85,B 0,C 180,E1 -683.417,E2 -683.417} C_VEL
LIN {X 0,Y 601.437,Z 365.57,A -85,B 0,C 180,E1 -686.064,E2 -686.064} C_VEL
LIN {X 0,Y 601.424,Z 365.566,A -85,B 0,C 180,E1 -688.546,E2 -688.546} C_VEL
LIN {X 0,Y 601.428,Z 365.568,A -85,B 0,C 180,E1 -691.373,E2 -691.373} C_VEL
LIN {X 0,Y 601.401,Z 365.569,A -85,B 0,C 180,E1 -693.636,E2 -693.636} C_VEL
LIN {X 0,Y 601.463,Z 365.564,A -85,B 0,C 180,E1 -695.86,E2 -695.86} C_VEL
LIN {X 0,Y 601.408,Z 365.568,A -85,B 0,C 180,E1 -698.761,E2 -698.761} C_VEL
LIN {X 0,Y 601.421,Z 365.57,A -85,B 0,C 180,E1 -701.608,E2 -701.608} C_VEL
LIN {X 0,Y 601.414,Z 365.57,A -85,B 0,C 180,E1 -704.409,E2 -704.409} C_VEL
LIN {X 0,Y 601.422,Z 365.566,A -85,B 0,C 180,E1 -707.172,E2 -707.172} C_VEL
LIN {X 0,Y 601.434,Z 365.572,A -85,B 0,C 180,E1 -709.905,E2 -709.905} C_VEL
LIN {X 0,Y 601.443,Z 365.564,A -85,B 0,C 180,E1 -712.615,E2 -712.615} C_VEL
LIN {X 0,Y 601.426,Z 365.569,A -85,B 0,C 180,E1 -715.308,E2 -715.308} C_VEL
LIN {X 0,Y 601.421,Z 365.568,A -85,B 0,C 180,E1 -717.991,E2 -717.991} C_VEL
LIN {X 0,Y 601.451,Z 365.563,A -85,B 0,C 180,E1 -720.669,E2 -720.669} C_VEL
LIN {X 0,Y 601.43,Z 365.57,A -85,B 0,C 180,E1 -723.35,E2 -723.35} C_VEL
LIN {X 0,Y 601.409,Z 365.568,A -85,B 0,C 180,E1 -726.037,E2 -726.037} C_VEL
LIN {X 0,Y 601.444,Z 365.57,A -85,B 0,C 180,E1 -728.738,E2 -728.738} C_VEL
LIN {X 0,Y 601.437,Z 365.565,A -85,B 0,C 180,E1 -731.458,E2 -731.458} C_VEL
LIN {X 0,Y 601.425,Z 365.568,A -85,B 0,C 180,E1 -734.205,E2 -734.205} C_VEL
LIN {X 0,Y 601.418,Z 365.571,A -85,B 0,C 180,E1 -736.986,E2 -736.986} C_VEL
LIN {X 0,Y 601.41,Z 365.568,A -85,B 0,C 180,E1 -739.809,E2 -739.809} C_VEL
LIN {X 0,Y 601.417,Z 365.57,A -85,B 0,C 180,E1 -742.683,E2 -742.683} C_VEL
LIN {X 0,Y 601.404,Z 365.568,A -85,B 0,C 180,E1 -744.879,E2 -744.879} C_VEL
LIN {X 0,Y 601.425,Z 365.572,A -85,B 0,C 180,E1 -747.363,E2 -747.363} C_VEL
LIN {X 0,Y 601.434,Z 365.565,A -85,B 0,C 180,E1 -750.164,E2 -750.164} C_VEL
LIN {X 0,Y 601.426,Z 365.572,A -85,B 0,C 180,E1 -752.715,E2 -752.715} C_VEL
LIN {X 0,Y 601.4,Z 365.569,A -85,B 0,C 180,E1 -755.112,E2 -755.112} C_VEL
LIN {X 0,Y 601.437,Z 365.567,A -85,B 0,C 180,E1 -757.419,E2 -757.419} C_VEL
LIN {X 0,Y 601.416,Z 365.568,A -85,B 0,C 180,E1 -759.995,E2 -759.995} C_VEL
LIN {X 0,Y 601.412,Z 365.572,A -85,B 0,C 180,E1 -762.67,E2 -762.67} C_VEL
LIN {X 0,Y 601.431,Z 365.565,A -85,B 0,C 180,E1 -765.482,E2 -765.482} C_VEL
LIN {X 0,Y 601.429,Z 365.568,A -85,B 0,C 180,E1 -768.407,E2 -768.407} C_VEL
LIN {X 0,Y 601.432,Z 365.572,A -85,B 0,C 180,E1 -771.529,E2 -771.529} C_VEL
LIN {X 0,Y 601.454,Z 365.684,A -85,B 0,C 180,E1 -774.16,E2 -774.16} C_VEL
LIN {X 0,Y 601.584,Z 372.843,A -85,B 0,C 180,E1 -776.371,E2 -776.371} C_VEL
LIN {X 0,Y 601.534,Z 381.859,A -85,B 0,C 180,E1 -779.064,E2 -779.064} C_VEL
LIN {X 0,Y 601.503,Z 391.126,A -85,B 0,C 180,E1 -781.757,E2 -781.757} C_VEL
LIN {X 0,Y 601.478,Z 400.394,A -85,B 0,C 180,E1 -784.384,E2 -784.384} C_VEL
LIN {X 0,Y 601.429,Z 409.661,A -85,B 0,C 180,E1 -786.954,E2 -786.954} C_VEL
LIN {X 0,Y 601.425,Z 420.252,A -85,B 0,C 180,E1 -789.835,E2 -789.835} C_VEL
LIN {X 0,Y 601.39,Z 430.844,A -85,B 0,C 180,E1 -792.662,E2 -792.662} C_VEL
LIN {X 0,Y 601.392,Z 441.435,A -85,B 0,C 180,E1 -795.448,E2 -795.448} C_VEL
LIN {X 0,Y 601.384,Z 451.53,A -85,B 0,C 180,E1 -798.071,E2 -798.071} C_VEL
LIN {X 0,Y 601.6,Z 464.175,A -85,B 0,C 180,E1 -798.331,E2 -798.331} C_VEL
LIN {X 0,Y 601.569,Z 476.165,A -85,B 0,C 180,E1 -798.686,E2 -798.686} C_VEL
LIN {X 0,Y 601.534,Z 487.965,A -85,B 0,C 180,E1 -799.167,E2 -799.167} C_VEL
LIN {X 0,Y 601.491,Z 500.165,A -85,B 0,C 180,E1 -799.821,E2 -799.821} C_VEL
LIN {X 0,Y 601.455,Z 511.401,A -85,B 0,C 180,E1 -800.585,E2 -800.585} C_VEL
LIN {X 0,Y 601.423,Z 521.335,A -85,B 0,C 180,E1 -801.431,E2 -801.431} C_VEL
LIN {X 0,Y 601.418,Z 530.959,A -85,B 0,C 180,E1 -802.446,E2 -802.446} C_VEL
LIN {X 0,Y 601.37,Z 538.224,A -85,B 0,C 180,E1 -803.398,E2 -803.398} C_VEL
LIN {X 0,Y 601.372,Z 543.865,A -85,B 0,C 180,E1 -804.299,E2 -804.299} C_VEL
LIN {X 0,Y 601.336,Z 548.95,A -85,B 0,C 180,E1 -805.307,E2 -805.307} C_VEL
LIN {X 0,Y 601.367,Z 552.896,A -85,B 0,C 180,E1 -806.315,E2 -806.315} C_VEL
LIN {X 0,Y 601.325,Z 555.809,A -85,B 0,C 180,E1 -807.32,E2 -807.32} C_VEL
LIN {X 0,Y 601.343,Z 557.201,A -85,B 0,C 180,E1 -807.991,E2 -807.991} C_VEL
LIN {X 0,Y 601.339,Z 558.784,A -85,B 0,C 180,E1 -809.33,E2 -809.33} C_VEL
LIN {X 0,Y 601.335,Z 559,A -85,B 0,C 180,E1 -810,E2 -810} C_VEL
LIN {X 0,Y 601.348,Z 558.184,A -85,B 0,C 180,E1 -811.339,E2 -811.339} C_VEL
LIN {X 0,Y 601.343,Z 557.202,A -85,B 0,C 180,E1 -812.009,E2 -812.009} C_VEL
LIN {X 0,Y 601.325,Z 555.809,A -85,B 0,C 180,E1 -812.68,E2 -812.68} C_VEL
LIN {X 0,Y 601.367,Z 552.896,A -85,B 0,C 180,E1 -813.685,E2 -813.685} C_VEL
LIN {X 0,Y 601.336,Z 548.95,A -85,B 0,C 180,E1 -814.693,E2 -814.693} C_VEL
LIN {X 0,Y 601.372,Z 542.877,A -85,B 0,C 180,E1 -815.869,E2 -815.869} C_VEL
LIN {X 0,Y 601.382,Z 536.235,A -85,B 0,C 180,E1 -816.88,E2 -816.88} C_VEL
LIN {X 0,Y 601.4,Z 527.989,A -85,B 0,C 180,E1 -817.892,E2 -817.892} C_VEL
LIN {X 0,Y 601.436,Z 519.536,A -85,B 0,C 180,E1 -818.738,E2 -818.738} C_VEL
LIN {X 0,Y 601.451,Z 509.091,A -85,B 0,C 180,E1 -819.585,E2 -819.585} C_VEL
LIN {X 0,Y 601.469,Z 498.756,A -85,B 0,C 180,E1 -820.264,E2 -820.264} C_VEL
LIN {X 0,Y 601.534,Z 487.917,A -85,B 0,C 180,E1 -820.835,E2 -820.835} C_VEL
LIN {X 0,Y 601.564,Z 475.385,A -85,B 0,C 180,E1 -821.34,E2 -821.34} C_VEL
LIN {X 0,Y 601.615,Z 462.352,A -85,B 0,C 180,E1 -821.711,E2 -821.711} C_VEL
LIN {X 0,Y 601.384,Z 451.53,A -85,B 0,C 180,E1 -821.929,E2 -821.929} C_VEL
LIN {X 0,Y 601.392,Z 441.435,A -85,B 0,C 180,E1 -824.552,E2 -824.552} C_VEL
LIN {X 0,Y 601.39,Z 430.844,A -85,B 0,C 180,E1 -827.338,E2 -827.338} C_VEL
LIN {X 0,Y 601.425,Z 420.253,A -85,B 0,C 180,E1 -830.165,E2 -830.165} C_VEL
LIN {X 0,Y 601.429,Z 409.662,A -85,B 0,C 180,E1 -833.046,E2 -833.046} C_VEL
LIN {X 0,Y 601.478,Z 400.394,A -85,B 0,C 180,E1 -835.616,E2 -835.616} C_VEL
LIN {X 0,Y 601.503,Z 391.127,A -85,B 0,C 180,E1 -838.243,E2 -838.243} C_VEL
LIN {X 0,Y 601.534,Z 381.859,A -85,B 0,C 180,E1 -840.936,E2 -840.936} C_VEL
LIN {X 0,Y 601.584,Z 372.844,A -85,B 0,C 180,E1 -843.629,E2 -843.629} C_VEL
LIN {X 0,Y 601.493,Z 365.973,A -85,B 0,C 180,E1 -845.748,E2 -845.748} C_VEL
LIN {X 0,Y 601.424,Z 365.57,A -85,B 0,C 180,E1 -845.932,E2 -845.932} C_VEL
LIN {X 0,Y 601.431,Z 365.572,A -85,B 0,C 180,E1 -848.47,E2 -848.47} C_VEL
LIN {X 0,Y 601.428,Z 365.568,A -85,B 0,C 180,E1 -851.593,E2 -851.593} C_VEL
LIN {X 0,Y 601.428,Z 365.566,A -85,B 0,C 180,E1 -854.535,E2 -854.535} C_VEL
LIN {X 0,Y 601.411,Z 365.571,A -85,B 0,C 180,E1 -857.41,E2 -857.41} C_VEL
LIN {X 0,Y 601.444,Z 365.57,A -85,B 0,C 180,E1 -860.464,E2 -860.464} C_VEL
LIN {X 0,Y 601.409,Z 365.569,A -85,B 0,C 180,E1 -863.417,E2 -863.417} C_VEL
LIN {X 0,Y 601.436,Z 365.567,A -85,B 0,C 180,E1 -866.064,E2 -866.064} C_VEL
LIN {X 0,Y 601.423,Z 365.567,A -85,B 0,C 180,E1 -868.545,E2 -868.545} C_VEL
LIN {X 0,Y 601.428,Z 365.566,A -85,B 0,C 180,E1 -871.373,E2 -871.373} C_VEL
LIN {X 0,Y 601.405,Z 365.569,A -85,B 0,C 180,E1 -873.636,E2 -873.636} C_VEL
LIN {X 0,Y 601.463,Z 365.567,A -85,B 0,C 180,E1 -875.86,E2 -875.86} C_VEL
LIN {X 0,Y 601.406,Z 365.569,A -85,B 0,C 180,E1 -878.761,E2 -878.761} C_VEL
LIN {X 0,Y 601.421,Z 365.567,A -85,B 0,C 180,E1 -881.608,E2 -881.608} C_VEL
LIN {X 0,Y 601.417,Z 365.573,A -85,B 0,C 180,E1 -884.409,E2 -884.409} C_VEL
LIN {X 0,Y 601.423,Z 365.566,A -85,B 0,C 180,E1 -887.172,E2 -887.172} C_VEL
LIN {X 0,Y 601.429,Z 365.569,A -85,B 0,C 180,E1 -889.905,E2 -889.905} C_VEL
LIN {X 0,Y 601.443,Z 365.565,A -85,B 0,C 180,E1 -892.615,E2 -892.615} C_VEL
LIN {X 0,Y 601.426,Z 365.567,A -85,B 0,C 180,E1 -895.308,E2 -895.308} C_VEL
LIN {X 0,Y 601.431,Z 365.569,A -85,B 0,C 180,E1 -897.991,E2 -897.991} C_VEL
LIN {X 0,Y 601.449,Z 365.563,A -85,B 0,C 180,E1 -900.67,E2 -900.67} C_VEL
LIN {X 0,Y 601.428,Z 365.573,A -85,B 0,C 180,E1 -903.35,E2 -903.35} C_VEL
LIN {X 0,Y 601.408,Z 365.568,A -85,B 0,C 180,E1 -906.037,E2 -906.037} C_VEL
LIN {X 0,Y 601.421,Z 365.57,A -85,B 0,C 180,E1 -908.738,E2 -908.738} C_VEL
LIN {X 0,Y 601.438,Z 365.566,A -85,B 0,C 180,E1 -911.458,E2 -911.458} C_VEL
LIN {X 0,Y 601.411,Z 365.569,A -85,B 0,C 180,E1 -912.375,E2 -912.375} C_VEL
LIN {X 0,Y 600.746,Z 365.651,A -85,B 0,C 180,E1 -912.934,E2 -912.934} C_VEL
LIN {X 0,Y 597.895,Z 366.01,A -85,B 0,C 180,E1 -913.842,E2 -913.842} C_VEL
LIN {X 0,Y 595.485,Z 366.311,A -85,B 0,C 180,E1 -914.572,E2 -914.572} C_VEL
LIN {X 0,Y 594.447,Z 366.44,A -85,B 0,C 180,E1 -915.136,E2 -915.136} C_VEL
LIN {X 0,Y 594.361,Z 366.448,A -85,B 0,C 180,E1 -915.327,E2 -915.327} C_VEL
LIN {X 0,Y 594.387,Z 366.448,A -85,B 0,C 180,E1 -917.194,E2 -917.194} C_VEL
LIN {X 0,Y 594.381,Z 366.445,A -85,B 0,C 180,E1 -920.054,E2 -920.054} C_VEL
LIN {X 0,Y 594.362,Z 366.445,A -85,B 0,C 180,E1 -922.968,E2 -922.968} C_VEL
LIN {X 0,Y 594.382,Z 366.445,A -85,B 0,C 180,E1 -925.193,E2 -925.193} C_VEL
LIN {X 0,Y 594.39,Z 366.447,A -85,B 0,C 180,E1 -927.527,E2 -927.527} C_VEL
LIN {X 0,Y 594.39,Z 366.444,A -85,B 0,C 180,E1 -930.328,E2 -930.328} C_VEL
LIN {X 0,Y 594.381,Z 366.444,A -85,B 0,C 180,E1 -932.95,E2 -932.95} C_VEL
LIN {X 0,Y 594.355,Z 366.448,A -85,B 0,C 180,E1 -935.409,E2 -935.409} C_VEL
LIN {X 0,Y 594.389,Z 366.445,A -85,B 0,C 180,E1 -937.941,E2 -937.941} C_VEL
LIN {X 0,Y 594.379,Z 366.449,A -85,B 0,C 180,E1 -940.822,E2 -940.822} C_VEL
LIN {X 0,Y 594.369,Z 366.446,A -85,B 0,C 180,E1 -943.3,E2 -943.3} C_VEL
LIN {X 0,Y 594.387,Z 366.45,A -85,B 0,C 180,E1 -946.159,E2 -946.159} C_VEL
LIN {X 0,Y 594.38,Z 366.445,A -85,B 0,C 180,E1 -949.178,E2 -949.178} C_VEL
LIN {X 0,Y 594.388,Z 366.442,A -85,B 0,C 180,E1 -952.059,E2 -952.059} C_VEL
LIN {X 0,Y 594.319,Z 366.458,A -85,B 0,C 180,E1 -954.681,E2 -954.681} C_VEL
LIN {X 0,Y 594.303,Z 367.83,A -85,B 0,C 180,E1 -956.234,E2 -956.234} C_VEL
LIN {X 0,Y 594.303,Z 370.553,A -85,B 0,C 180,E1 -958.646,E2 -958.646} C_VEL
LIN {X 0,Y 594.291,Z 373.29,A -85,B 0,C 180,E1 -961.059,E2 -961.059} C_VEL
LIN {X 0,Y 594.297,Z 376.962,A -85,B 0,C 180,E1 -964.052,E2 -964.052} C_VEL
LIN {X 0,Y 594.239,Z 379.844,A -85,B 0,C 180,E1 -966.29,E2 -966.29} C_VEL
LIN {X 0,Y 594.296,Z 383.687,A -85,B 0,C 180,E1 -969.22,E2 -969.22} C_VEL
LIN {X 0,Y 594.212,Z 387.53,A -85,B 0,C 180,E1 -972.091,E2 -972.091} C_VEL
LIN {X 0,Y 594.245,Z 390.413,A -85,B 0,C 180,E1 -974.216,E2 -974.216} C_VEL
LIN {X 0,Y 594.236,Z 394.257,A -85,B 0,C 180,E1 -977.014,E2 -977.014} C_VEL
LIN {X 0,Y 594.271,Z 395.668,A -85,B 0,C 180,E1 -978.034,E2 -978.034} C_VEL
LIN {X 0,Y 594.654,Z 400.446,A -85,B 0,C 180,E1 -978.15,E2 -978.15} C_VEL
LIN {X 0,Y 594.596,Z 413.04,A -85,B 0,C 180,E1 -978.492,E2 -978.492} C_VEL
LIN {X 0,Y 594.559,Z 424.865,A -85,B 0,C 180,E1 -978.944,E2 -978.944} C_VEL
LIN {X 0,Y 594.5,Z 436.524,A -85,B 0,C 180,E1 -979.528,E2 -979.528} C_VEL
LIN {X 0,Y 594.448,Z 447.316,A -85,B 0,C 180,E1 -980.215,E2 -980.215} C_VEL
LIN {X 0,Y 594.404,Z 457.091,A -85,B 0,C 180,E1 -980.987,E2 -980.987} C_VEL
LIN {X 0,Y 594.366,Z 465.986,A -85,B 0,C 180,E1 -981.843,E2 -981.843} C_VEL
LIN {X 0,Y 594.345,Z 474.672,A -85,B 0,C 180,E1 -982.868,E2 -982.868} C_VEL
LIN {X 0,Y 594.29,Z 481.6,A -85,B 0,C 180,E1 -983.89,E2 -983.89} C_VEL
LIN {X 0,Y 594.253,Z 487.152,A -85,B 0,C 180,E1 -984.911,E2 -984.911} C_VEL
LIN {X 0,Y 594.263,Z 491.513,A -85,B 0,C 180,E1 -985.931,E2 -985.931} C_VEL
LIN {X 0,Y 594.267,Z 493.817,A -85,B 0,C 180,E1 -986.61,E2 -986.61} C_VEL
LIN {X 0,Y 594.225,Z 495.695,A -85,B 0,C 180,E1 -987.288,E2 -987.288} C_VEL
LIN {X 0,Y 594.242,Z 497.127,A -85,B 0,C 180,E1 -987.967,E2 -987.967} C_VEL
LIN {X 0,Y 594.24,Z 498.753,A -85,B 0,C 180,E1 -989.322,E2 -989.322} C_VEL
LIN {X 0,Y 594.236,Z 498.996,A -85,B 0,C 180,E1 -990,E2 -990} C_VEL
LIN {X 0,Y 594.239,Z 498.815,A -85,B 0,C 180,E1 -990.678,E2 -990.678} C_VEL
LIN {X 0,Y 594.242,Z 497.275,A -85,B 0,C 180,E1 -992.033,E2 -992.033} C_VEL
LIN {X 0,Y 594.226,Z 495.915,A -85,B 0,C 180,E1 -992.712,E2 -992.712} C_VEL
LIN {X 0,Y 594.289,Z 493.038,A -85,B 0,C 180,E1 -993.729,E2 -993.729} C_VEL
LIN {X 0,Y 594.241,Z 489.138,A -85,B 0,C 180,E1 -994.749,E2 -994.749} C_VEL
LIN {X 0,Y 594.3,Z 484.106,A -85,B 0,C 180,E1 -995.769,E2 -995.769} C_VEL
LIN {X 0,Y 594.316,Z 477.787,A -85,B 0,C 180,E1 -996.791,E2 -996.791} C_VEL
LIN {X 0,Y 594.346,Z 469.868,A -85,B 0,C 180,E1 -997.816,E2 -997.816} C_VEL
LIN {X 0,Y 594.381,Z 460.022,A -85,B 0,C 180,E1 -998.842,E2 -998.842} C_VEL
LIN {X 0,Y 594.435,Z 449.7,A -85,B 0,C 180,E1 -999.699,E2 -999.699} C_VEL
LIN {X 0,Y 594.5,Z 438.076,A -85,B 0,C 180,E1 -1000.472,E2 -1000.472} C_VEL
LIN {X 0,Y 594.548,Z 426.18,A -85,B 0,C 180,E1 -1001.089,E2 -1001.089} C_VEL
LIN {X 0,Y 594.589,Z 413.226,A -85,B 0,C 180,E1 -1001.592,E2 -1001.592} C_VEL
LIN {X 0,Y 594.66,Z 400.591,A -85,B 0,C 180,E1 -1001.936,E2 -1001.936} C_VEL
LIN {X 0,Y 594.272,Z 395.672,A -85,B 0,C 180,E1 -1002.053,E2 -1002.053} C_VEL
LIN {X 0,Y 594.237,Z 392.458,A -85,B 0,C 180,E1 -1004.381,E2 -1004.381} C_VEL
LIN {X 0,Y 594.241,Z 388.613,A -85,B 0,C 180,E1 -1007.198,E2 -1007.198} C_VEL
LIN {X 0,Y 594.243,Z 385.729,A -85,B 0,C 180,E1 -1009.339,E2 -1009.339} C_VEL
LIN {X 0,Y 594.225,Z 382.845,A -85,B 0,C 180,E1 -1011.509,E2 -1011.509} C_VEL
LIN {X 0,Y 594.278,Z 378.999,A -85,B 0,C 180,E1 -1014.451,E2 -1014.451} C_VEL
LIN {X 0,Y 594.266,Z 376.115,A -85,B 0,C 180,E1 -1016.706,E2 -1016.706} C_VEL
LIN {X 0,Y 594.273,Z 373.303,A -85,B 0,C 180,E1 -1019.005,E2 -1019.005} C_VEL
LIN {X 0,Y 594.308,Z 370.355,A -85,B 0,C 180,E1 -1021.631,E2 -1021.631} C_VEL
LIN {X 0,Y 594.298,Z 367.012,A -85,B 0,C 180,E1 -1024.586,E2 -1024.586} C_VEL
LIN {X 0,Y 594.323,Z 366.458,A -85,B 0,C 180,E1 -1025.411,E2 -1025.411} C_VEL
LIN {X 0,Y 594.389,Z 366.442,A -85,B 0,C 180,E1 -1027.941,E2 -1027.941} C_VEL
LIN {X 0,Y 594.381,Z 366.446,A -85,B 0,C 180,E1 -1030.822,E2 -1030.822} C_VEL
LIN {X 0,Y 594.388,Z 366.449,A -85,B 0,C 180,E1 -1033.841,E2 -1033.841} C_VEL
LIN {X 0,Y 594.369,Z 366.445,A -85,B 0,C 180,E1 -1036.7,E2 -1036.7} C_VEL
LIN {X 0,Y 594.369,Z 366.448,A -85,B 0,C 180,E1 -1039.433,E2 -1039.433} C_VEL
LIN {X 0,Y 594.394,Z 366.448,A -85,B 0,C 180,E1 -1042.392,E2 -1042.392} C_VEL
LIN {X 0,Y 594.399,Z 366.442,A -85,B 0,C 180,E1 -1045.421,E2 -1045.421} C_VEL
LIN {X 0,Y 594.382,Z 366.443,A -85,B 0,C 180,E1 -1048.358,E2 -1048.358} C_VEL
LIN {X 0,Y 594.386,Z 366.45,A -85,B 0,C 180,E1 -1051.043,E2 -1051.043} C_VEL
LIN {X 0,Y 594.387,Z 366.443,A -85,B 0,C 180,E1 -1053.3,E2 -1053.3} C_VEL
LIN {X 0,Y 594.383,Z 366.449,A -85,B 0,C 180,E1 -1056.296,E2 -1056.296} C_VEL
LIN {X 0,Y 594.409,Z 366.442,A -85,B 0,C 180,E1 -1059.224,E2 -1059.224} C_VEL
LIN {X 0,Y 594.356,Z 366.446,A -85,B 0,C 180,E1 -1062.095,E2 -1062.095} C_VEL
LIN {X 0,Y 594.367,Z 366.446,A -85,B 0,C 180,E1 -1064.219,E2 -1064.219} C_VEL
LIN {X 0,Y 594.385,Z 366.449,A -85,B 0,C 180,E1 -1066.321,E2 -1066.321} C_VEL
LIN {X 0,Y 594.376,Z 366.444,A -85,B 0,C 180,E1 -1069.095,E2 -1069.095} C_VEL
LIN {X 0,Y 594.385,Z 366.446,A -85,B 0,C 180,E1 -1071.843,E2 -1071.843} C_VEL
LIN {X 0,Y 594.366,Z 366.446,A -85,B 0,C 180,E1 -1073.891,E2 -1073.891} C_VEL
LIN {X 0,Y 594.379,Z 366.45,A -85,B 0,C 180,E1 -1076.611,E2 -1076.611} C_VEL
LIN {X 0,Y 594.421,Z 366.438,A -85,B 0,C 180,E1 -1079.323,E2 -1079.323} C_VEL
LIN {X 0,Y 594.403,Z 366.445,A -85,B 0,C 180,E1 -1082.033,E2 -1082.033} C_VEL
LIN {X 0,Y 594.398,Z 366.442,A -85,B 0,C 180,E1 -1084.748,E2 -1084.748} C_VEL
LIN {X 0,Y 594.398,Z 366.442,A -85,B 0,C 180,E1 -1087.473,E2 -1087.473} C_VEL
LIN {X 0,Y 594.39,Z 366.448,A -85,B 0,C 180,E1 -1090.216,E2 -1090.216} C_VEL
LIN {X 0,Y 594.371,Z 366.444,A -85,B 0,C 180,E1 -1092.983,E2 -1092.983} C_VEL
LIN {X 0,Y 594.375,Z 366.446,A -85,B 0,C 180,E1 -1095.078,E2 -1095.078} C_VEL
LIN {X 0,Y 594.384,Z 366.45,A -85,B 0,C 180,E1 -1097.194,E2 -1097.194} C_VEL
LIN {X 0,Y 594.38,Z 366.444,A -85,B 0,C 180,E1 -1100.054,E2 -1100.054} C_VEL
LIN {X 0,Y 594.361,Z 366.446,A -85,B 0,C 180,E1 -1102.967,E2 -1102.967} C_VEL
LIN {X 0,Y 594.378,Z 366.444,A -85,B 0,C 180,E1 -1105.193,E2 -1105.193} C_VEL
LIN {X 0,Y 594.391,Z 366.449,A -85,B 0,C 180,E1 -1107.527,E2 -1107.527} C_VEL
LIN {X 0,Y 594.391,Z 366.443,A -85,B 0,C 180,E1 -1110.328,E2 -1110.328} C_VEL
LIN {X 0,Y 594.382,Z 366.446,A -85,B 0,C 180,E1 -1112.95,E2 -1112.95} C_VEL
LIN {X 0,Y 594.355,Z 366.447,A -85,B 0,C 180,E1 -1115.409,E2 -1115.409} C_VEL
LIN {X 0,Y 594.387,Z 366.447,A -85,B 0,C 180,E1 -1117.941,E2 -1117.941} C_VEL
LIN {X 0,Y 594.38,Z 366.446,A -85,B 0,C 180,E1 -1120.822,E2 -1120.822} C_VEL
LIN {X 0,Y 594.372,Z 366.445,A -85,B 0,C 180,E1 -1123.839,E2 -1123.839} C_VEL
LIN {X 0,Y 594.384,Z 366.445,A -85,B 0,C 180,E1 -1126.702,E2 -1126.702} C_VEL
LIN {X 0,Y 594.37,Z 366.449,A -85,B 0,C 180,E1 -1129.433,E2 -1129.433} C_VEL
LIN {X 0,Y 594.392,Z 366.443,A -85,B 0,C 180,E1 -1132.392,E2 -1132.392} C_VEL
LIN {X 0,Y 594.398,Z 366.634,A -85,B 0,C 180,E1 -1133.968,E2 -1133.968} C_VEL
LIN {X 0,Y 594.64,Z 371.268,A -85,B 0,C 180,E1 -1135.437,E2 -1135.437} C_VEL
LIN {X 0,Y 594.609,Z 379.211,A -85,B 0,C 180,E1 -1137.867,E2 -1137.867} C_VEL
LIN {X 0,Y 594.565,Z 388.478,A -85,B 0,C 180,E1 -1140.623,E2 -1140.623} C_VEL
LIN {X 0,Y 594.506,Z 397.746,A -85,B 0,C 180,E1 -1143.306,E2 -1143.306} C_VEL
LIN {X 0,Y 594.45,Z 408.337,A -85,B 0,C 180,E1 -1146.298,E2 -1146.298} C_VEL
LIN {X 0,Y 594.408,Z 418.928,A -85,B 0,C 180,E1 -1149.224,E2 -1149.224} C_VEL
LIN {X 0,Y 594.359,Z 429.52,A -85,B 0,C 180,E1 -1152.095,E2 -1152.095} C_VEL
LIN {X 0,Y 594.325,Z 440.111,A -85,B 0,C 180,E1 -1154.921,E2 -1154.921} C_VEL
LIN {X 0,Y 594.299,Z 450.702,A -85,B 0,C 180,E1 -1157.71,E2 -1157.71} C_VEL
LIN {X 0,Y 594.299,Z 451.53,A -85,B 0,C 180,E1 -1157.926,E2 -1157.926} C_VEL
LIN {X 0,Y 594.678,Z 457.222,A -85,B 0,C 180,E1 -1158.042,E2 -1158.042} C_VEL
LIN {X 0,Y 594.641,Z 470.49,A -85,B 0,C 180,E1 -1158.366,E2 -1158.366} C_VEL
LIN {X 0,Y 594.589,Z 482.318,A -85,B 0,C 180,E1 -1158.788,E2 -1158.788} C_VEL
LIN {X 0,Y 594.514,Z 494.205,A -85,B 0,C 180,E1 -1159.356,E2 -1159.356} C_VEL
LIN {X 0,Y 594.475,Z 505.473,A -85,B 0,C 180,E1 -1160.043,E2 -1160.043} C_VEL
LIN {X 0,Y 594.406,Z 515.645,A -85,B 0,C 180,E1 -1160.815,E2 -1160.815} C_VEL
LIN {X 0,Y 594.372,Z 524.786,A -85,B 0,C 180,E1 -1161.671,E2 -1161.671} C_VEL
LIN {X 0,Y 594.317,Z 533.69,A -85,B 0,C 180,E1 -1162.697,E2 -1162.697} C_VEL
LIN {X 0,Y 594.281,Z 540.169,A -85,B 0,C 180,E1 -1163.615,E2 -1163.615} C_VEL
LIN {X 0,Y 594.289,Z 545.68,A -85,B 0,C 180,E1 -1164.571,E2 -1164.571} C_VEL
LIN {X 0,Y 594.27,Z 550.371,A -85,B 0,C 180,E1 -1165.591,E2 -1165.591} C_VEL
LIN {X 0,Y 594.267,Z 553.956,A -85,B 0,C 180,E1 -1166.61,E2 -1166.61} C_VEL
LIN {X 0,Y 594.226,Z 555.809,A -85,B 0,C 180,E1 -1167.288,E2 -1167.288} C_VEL
LIN {X 0,Y 594.242,Z 557.201,A -85,B 0,C 180,E1 -1167.967,E2 -1167.967} C_VEL
LIN {X 0,Y 594.239,Z 558.784,A -85,B 0,C 180,E1 -1169.322,E2 -1169.322} C_VEL
LIN {X 0,Y 594.236,Z 559,A -85,B 0,C 180,E1 -1170,E2 -1170} C_VEL
LIN {X 0,Y 594.248,Z 558.184,A -85,B 0,C 180,E1 -1171.355,E2 -1171.355} C_VEL
LIN {X 0,Y 594.242,Z 557.202,A -85,B 0,C 180,E1 -1172.033,E2 -1172.033} C_VEL
LIN {X 0,Y 594.226,Z 555.809,A -85,B 0,C 180,E1 -1172.712,E2 -1172.712} C_VEL
LIN {X 0,Y 594.288,Z 552.896,A -85,B 0,C 180,E1 -1173.729,E2 -1173.729} C_VEL
LIN {X 0,Y 594.241,Z 548.95,A -85,B 0,C 180,E1 -1174.749,E2 -1174.749} C_VEL
LIN {X 0,Y 594.304,Z 542.877,A -85,B 0,C 180,E1 -1175.939,E2 -1175.939} C_VEL
LIN {X 0,Y 594.308,Z 536.236,A -85,B 0,C 180,E1 -1176.962,E2 -1176.962} C_VEL
LIN {X 0,Y 594.359,Z 527.989,A -85,B 0,C 180,E1 -1177.986,E2 -1177.986} C_VEL
LIN {X 0,Y 594.382,Z 519.537,A -85,B 0,C 180,E1 -1178.842,E2 -1178.842} C_VEL
LIN {X 0,Y 594.435,Z 509.092,A -85,B 0,C 180,E1 -1179.699,E2 -1179.699} C_VEL
LIN {X 0,Y 594.482,Z 498.757,A -85,B 0,C 180,E1 -1180.386,E2 -1180.386} C_VEL
LIN {X 0,Y 594.557,Z 487.732,A -85,B 0,C 180,E1 -1180.973,E2 -1180.973} C_VEL
LIN {X 0,Y 594.59,Z 475.712,A -85,B 0,C 180,E1 -1181.464,E2 -1181.464} C_VEL
LIN {X 0,Y 594.653,Z 462.351,A -85,B 0,C 180,E1 -1181.85,E2 -1181.85} C_VEL
LIN {X 0,Y 594.467,Z 452.861,A -85,B 0,C 180,E1 -1182.038,E2 -1182.038} C_VEL
LIN {X 0,Y 594.299,Z 451.53,A -85,B 0,C 180,E1 -1182.074,E2 -1182.074} C_VEL
LIN {X 0,Y 594.319,Z 441.435,A -85,B 0,C 180,E1 -1184.729,E2 -1184.729} C_VEL
LIN {X 0,Y 594.336,Z 430.844,A -85,B 0,C 180,E1 -1187.55,E2 -1187.55} C_VEL
LIN {X 0,Y 594.384,Z 420.253,A -85,B 0,C 180,E1 -1190.415,E2 -1190.415} C_VEL
LIN {X 0,Y 594.438,Z 409.662,A -85,B 0,C 180,E1 -1193.333,E2 -1193.333} C_VEL
LIN {X 0,Y 594.495,Z 400.025,A -85,B 0,C 180,E1 -1196.044,E2 -1196.044} C_VEL
LIN {X 0,Y 594.51,Z 391.143,A -85,B 0,C 180,E1 -1198.6,E2 -1198.6} C_VEL
LIN {X 0,Y 594.589,Z 381.859,A -85,B 0,C 180,E1 -1201.338,E2 -1201.338} C_VEL
LIN {X 0,Y 594.612,Z 372.539,A -85,B 0,C 180,E1 -1204.171,E2 -1204.171} C_VEL
LIN {X 0,Y 594.53,Z 367.296,A -85,B 0,C 180,E1 -1205.813,E2 -1205.813} C_VEL
LIN {X 0,Y 594.373,Z 366.45,A -85,B 0,C 180,E1 -1206.138,E2 -1206.138} C_VEL
LIN {X 0,Y 594.379,Z 366.449,A -85,B 0,C 180,E1 -1208.806,E2 -1208.806} C_VEL
LIN {X 0,Y 594.388,Z 366.448,A -85,B 0,C 180,E1 -1211.849,E2 -1211.849} C_VEL
LIN {X 0,Y 594.386,Z 366.445,A -85,B 0,C 180,E1 -1214.236,E2 -1214.236} C_VEL
LIN {X 0,Y 594.362,Z 366.453,A -85,B 0,C 180,E1 -1217.149,E2 -1217.149} C_VEL
LIN {X 0,Y 594.37,Z 366.445,A -85,B 0,C 180,E1 -1219.433,E2 -1219.433} C_VEL
LIN {X 0,Y 594.392,Z 366.448,A -85,B 0,C 180,E1 -1222.392,E2 -1222.392} C_VEL
LIN {X 0,Y 594.385,Z 366.447,A -85,B 0,C 180,E1 -1225.42,E2 -1225.42} C_VEL
LIN {X 0,Y 594.381,Z 366.443,A -85,B 0,C 180,E1 -1228.357,E2 -1228.357} C_VEL
LIN {X 0,Y 594.385,Z 366.447,A -85,B 0,C 180,E1 -1231.043,E2 -1231.043} C_VEL
LIN {X 0,Y 594.389,Z 366.446,A -85,B 0,C 180,E1 -1233.977,E2 -1233.977} C_VEL
LIN {X 0,Y 594.381,Z 366.446,A -85,B 0,C 180,E1 -1236.296,E2 -1236.296} C_VEL
LIN {X 0,Y 594.407,Z 366.445,A -85,B 0,C 180,E1 -1239.224,E2 -1239.224} C_VEL
LIN {X 0,Y 594.355,Z 366.447,A -85,B 0,C 180,E1 -1242.095,E2 -1242.095} C_VEL
LIN {X 0,Y 594.37,Z 366.448,A -85,B 0,C 180,E1 -1244.219,E2 -1244.219} C_VEL
LIN {X 0,Y 594.389,Z 366.449,A -85,B 0,C 180,E1 -1246.321,E2 -1246.321} C_VEL
LIN {X 0,Y 594.376,Z 366.445,A -85,B 0,C 180,E1 -1249.095,E2 -1249.095} C_VEL
LIN {X 0,Y 594.418,Z 366.44,A -85,B 0,C 180,E1 -1251.843,E2 -1251.843} C_VEL
LIN {X 0,Y 594.395,Z 366.446,A -85,B 0,C 180,E1 -1254.572,E2 -1254.572} C_VEL
LIN {X 0,Y 594.411,Z 366.439,A -85,B 0,C 180,E1 -1257.289,E2 -1257.289} C_VEL
LIN {X 0,Y 594.416,Z 366.446,A -85,B 0,C 180,E1 -1260,E2 -1260} C_VEL
LIN {X 0,Y 594.41,Z 366.44,A -85,B 0,C 180,E1 -1262.711,E2 -1262.711} C_VEL
LIN {X 0,Y 594.398,Z 366.444,A -85,B 0,C 180,E1 -1265.428,E2 -1265.428} C_VEL
LIN {X 0,Y 594.397,Z 366.441,A -85,B 0,C 180,E1 -1267.473,E2 -1267.473} C_VEL
LIN {X 0,Y 594.392,Z 366.449,A -85,B 0,C 180,E1 -1270.216,E2 -1270.216} C_VEL
LIN {X 0,Y 594.369,Z 366.445,A -85,B 0,C 180,E1 -1272.983,E2 -1272.983} C_VEL
LIN {X 0,Y 594.361,Z 366.448,A -85,B 0,C 180,E1 -1275.327,E2 -1275.327} C_VEL
LIN {X 0,Y 593.685,Z 366.532,A -85,B 0,C 180,E1 -1275.893,E2 -1275.893} C_VEL
LIN {X 0,Y 590.815,Z 366.892,A -85,B 0,C 180,E1 -1276.811,E2 -1276.811} C_VEL
LIN {X 0,Y 588.404,Z 367.19,A -85,B 0,C 180,E1 -1277.549,E2 -1277.549} C_VEL
LIN {X 0,Y 587.382,Z 367.316,A -85,B 0,C 180,E1 -1278.119,E2 -1278.119} C_VEL
LIN {X 0,Y 587.307,Z 367.326,A -85,B 0,C 180,E1 -1278.312,E2 -1278.312} C_VEL
LIN {X 0,Y 587.335,Z 367.322,A -85,B 0,C 180,E1 -1281.038,E2 -1281.038} C_VEL
LIN {X 0,Y 587.32,Z 367.323,A -85,B 0,C 180,E1 -1283.259,E2 -1283.259} C_VEL
LIN {X 0,Y 587.338,Z 367.327,A -85,B 0,C 180,E1 -1285.517,E2 -1285.517} C_VEL
LIN {X 0,Y 587.35,Z 367.321,A -85,B 0,C 180,E1 -1287.818,E2 -1287.818} C_VEL
LIN {X 0,Y 587.341,Z 367.325,A -85,B 0,C 180,E1 -1290.51,E2 -1290.51} C_VEL
LIN {X 0,Y 587.337,Z 367.321,A -85,B 0,C 180,E1 -1293.397,E2 -1293.397} C_VEL
LIN {X 0,Y 587.296,Z 367.333,A -85,B 0,C 180,E1 -1295.9,E2 -1295.9} C_VEL
LIN {X 0,Y 587.336,Z 367.321,A -85,B 0,C 180,E1 -1298.479,E2 -1298.479} C_VEL
LIN {X 0,Y 587.339,Z 367.326,A -85,B 0,C 180,E1 -1301.157,E2 -1301.157} C_VEL
LIN {X 0,Y 587.315,Z 367.327,A -85,B 0,C 180,E1 -1304.112,E2 -1304.112} C_VEL
LIN {X 0,Y 587.325,Z 367.322,A -85,B 0,C 180,E1 -1306.994,E2 -1306.994} C_VEL
LIN {X 0,Y 587.316,Z 367.328,A -85,B 0,C 180,E1 -1309.746,E2 -1309.746} C_VEL
LIN {X 0,Y 587.349,Z 367.32,A -85,B 0,C 180,E1 -1312.392,E2 -1312.392} C_VEL
LIN {X 0,Y 587.257,Z 367.338,A -85,B 0,C 180,E1 -1314.939,E2 -1314.939} C_VEL
LIN {X 0,Y 587.245,Z 369.26,A -85,B 0,C 180,E1 -1316.903,E2 -1316.903} C_VEL
LIN {X 0,Y 587.228,Z 372.173,A -85,B 0,C 180,E1 -1319.509,E2 -1319.509} C_VEL
LIN {X 0,Y 587.197,Z 375.357,A -85,B 0,C 180,E1 -1322.337,E2 -1322.337} C_VEL
LIN {X 0,Y 587.177,Z 377.923,A -85,B 0,C 180,E1 -1324.476,E2 -1324.476} C_VEL
LIN {X 0,Y 587.151,Z 381.369,A -85,B 0,C 180,E1 -1327.171,E2 -1327.171} C_VEL
LIN {X 0,Y 587.167,Z 384.649,A -85,B 0,C 180,E1 -1329.689,E2 -1329.689} C_VEL
LIN {X 0,Y 587.132,Z 388.492,A -85,B 0,C 180,E1 -1332.587,E2 -1332.587} C_VEL
LIN {X 0,Y 587.137,Z 391.375,A -85,B 0,C 180,E1 -1334.732,E2 -1334.732} C_VEL
LIN {X 0,Y 587.138,Z 394.257,A -85,B 0,C 180,E1 -1336.854,E2 -1336.854} C_VEL
LIN {X 0,Y 587.161,Z 395.669,A -85,B 0,C 180,E1 -1337.887,E2 -1337.887} C_VEL
LIN {X 0,Y 587.706,Z 401.384,A -85,B 0,C 180,E1 -1338.03,E2 -1338.03} C_VEL
LIN {X 0,Y 587.623,Z 414.6,A -85,B 0,C 180,E1 -1338.406,E2 -1338.406} C_VEL
LIN {X 0,Y 587.576,Z 426.643,A -85,B 0,C 180,E1 -1338.889,E2 -1338.889} C_VEL
LIN {X 0,Y 587.504,Z 438.022,A -85,B 0,C 180,E1 -1339.489,E2 -1339.489} C_VEL
LIN {X 0,Y 587.43,Z 449.655,A -85,B 0,C 180,E1 -1340.271,E2 -1340.271} C_VEL
LIN {X 0,Y 587.344,Z 459.037,A -85,B 0,C 180,E1 -1341.051,E2 -1341.051} C_VEL
LIN {X 0,Y 587.3,Z 467.6,A -85,B 0,C 180,E1 -1341.917,E2 -1341.917} C_VEL
LIN {X 0,Y 587.262,Z 475.914,A -85,B 0,C 180,E1 -1342.954,E2 -1342.954} C_VEL
LIN {X 0,Y 587.218,Z 482.614,A -85,B 0,C 180,E1 -1343.989,E2 -1343.989} C_VEL
LIN {X 0,Y 587.146,Z 488.758,A -85,B 0,C 180,E1 -1345.194,E2 -1345.194} C_VEL
LIN {X 0,Y 587.213,Z 492.748,A -85,B 0,C 180,E1 -1346.226,E2 -1346.226} C_VEL
LIN {X 0,Y 587.131,Z 495.696,A -85,B 0,C 180,E1 -1347.256,E2 -1347.256} C_VEL
LIN {X 0,Y 587.141,Z 497.128,A -85,B 0,C 180,E1 -1347.942,E2 -1347.942} C_VEL
LIN {X 0,Y 587.14,Z 498.754,A -85,B 0,C 180,E1 -1349.314,E2 -1349.314} C_VEL
LIN {X 0,Y 587.137,Z 498.996,A -85,B 0,C 180,E1 -1350,E2 -1350} C_VEL
LIN {X 0,Y 587.14,Z 498.815,A -85,B 0,C 180,E1 -1350.686,E2 -1350.686} C_VEL
LIN {X 0,Y 587.141,Z 497.274,A -85,B 0,C 180,E1 -1352.058,E2 -1352.058} C_VEL
LIN {X 0,Y 587.133,Z 495.913,A -85,B 0,C 180,E1 -1352.744,E2 -1352.744} C_VEL
LIN {X 0,Y 587.213,Z 493.036,A -85,B 0,C 180,E1 -1353.774,E2 -1353.774} C_VEL
LIN {X 0,Y 587.147,Z 489.136,A -85,B 0,C 180,E1 -1354.806,E2 -1354.806} C_VEL
LIN {X 0,Y 587.23,Z 484.104,A -85,B 0,C 180,E1 -1355.839,E2 -1355.839} C_VEL
LIN {X 0,Y 587.23,Z 477.783,A -85,B 0,C 180,E1 -1356.874,E2 -1356.874} C_VEL
LIN {X 0,Y 587.288,Z 469.864,A -85,B 0,C 180,E1 -1357.91,E2 -1357.91} C_VEL
LIN {X 0,Y 587.343,Z 460.016,A -85,B 0,C 180,E1 -1358.949,E2 -1358.949} C_VEL
LIN {X 0,Y 587.422,Z 449.694,A -85,B 0,C 180,E1 -1359.816,E2 -1359.816} C_VEL
LIN {X 0,Y 587.497,Z 439.486,A -85,B 0,C 180,E1 -1360.511,E2 -1360.511} C_VEL
LIN {X 0,Y 587.567,Z 427.138,A -85,B 0,C 180,E1 -1361.179,E2 -1361.179} C_VEL
LIN {X 0,Y 587.616,Z 414.452,A -85,B 0,C 180,E1 -1361.69,E2 -1361.69} C_VEL
LIN {X 0,Y 587.715,Z 401.483,A -85,B 0,C 180,E1 -1362.058,E2 -1362.058} C_VEL
LIN {X 0,Y 587.292,Z 396.852,A -85,B 0,C 180,E1 -1362.162,E2 -1362.162} C_VEL
LIN {X 0,Y 587.161,Z 395.642,A -85,B 0,C 180,E1 -1362.223,E2 -1362.223} C_VEL
LIN {X 0,Y 587.129,Z 392.457,A -85,B 0,C 180,E1 -1364.559,E2 -1364.559} C_VEL
LIN {X 0,Y 587.147,Z 389.503,A -85,B 0,C 180,E1 -1366.748,E2 -1366.748} C_VEL
LIN {X 0,Y 587.136,Z 385.728,A -85,B 0,C 180,E1 -1369.582,E2 -1369.582} C_VEL
LIN {X 0,Y 587.143,Z 382.844,A -85,B 0,C 180,E1 -1371.782,E2 -1371.782} C_VEL
LIN {X 0,Y 587.18,Z 378.998,A -85,B 0,C 180,E1 -1374.767,E2 -1374.767} C_VEL
LIN {X 0,Y 587.17,Z 376.158,A -85,B 0,C 180,E1 -1377.054,E2 -1377.054} C_VEL
LIN {X 0,Y 587.234,Z 372.61,A -85,B 0,C 180,E1 -1380.176,E2 -1380.176} C_VEL
LIN {X 0,Y 587.245,Z 369.361,A -85,B 0,C 180,E1 -1383.097,E2 -1383.097} C_VEL
LIN {X 0,Y 587.259,Z 367.338,A -85,B 0,C 180,E1 -1385.061,E2 -1385.061} C_VEL
LIN {X 0,Y 587.349,Z 367.321,A -85,B 0,C 180,E1 -1387.608,E2 -1387.608} C_VEL
LIN {X 0,Y 587.317,Z 367.327,A -85,B 0,C 180,E1 -1390.255,E2 -1390.255} C_VEL
LIN {X 0,Y 587.326,Z 367.322,A -85,B 0,C 180,E1 -1393.006,E2 -1393.006} C_VEL
LIN {X 0,Y 587.316,Z 367.328,A -85,B 0,C 180,E1 -1395.888,E2 -1395.888} C_VEL
LIN {X 0,Y 587.339,Z 367.326,A -85,B 0,C 180,E1 -1398.925,E2 -1398.925} C_VEL
LIN {X 0,Y 587.337,Z 367.321,A -85,B 0,C 180,E1 -1401.521,E2 -1401.521} C_VEL
LIN {X 0,Y 587.299,Z 367.331,A -85,B 0,C 180,E1 -1404.1,E2 -1404.1} C_VEL
LIN {X 0,Y 587.338,Z 367.321,A -85,B 0,C 180,E1 -1406.603,E2 -1406.603} C_VEL
LIN {X 0,Y 587.342,Z 367.326,A -85,B 0,C 180,E1 -1409.49,E2 -1409.49} C_VEL
LIN {X 0,Y 587.356,Z 367.32,A -85,B 0,C 180,E1 -1412.307,E2 -1412.307} C_VEL
LIN {X 0,Y 587.357,Z 367.318,A -85,B 0,C 180,E1 -1415.242,E2 -1415.242} C_VEL
LIN {X 0,Y 587.324,Z 367.325,A -85,B 0,C 180,E1 -1418.226,E2 -1418.226} C_VEL
LIN {X 0,Y 587.354,Z 367.324,A -85,B 0,C 180,E1 -1421.151,E2 -1421.151} C_VEL
LIN {X 0,Y 587.322,Z 367.323,A -85,B 0,C 180,E1 -1424.025,E2 -1424.025} C_VEL
LIN {X 0,Y 587.363,Z 367.321,A -85,B 0,C 180,E1 -1426.154,E2 -1426.154} C_VEL
LIN {X 0,Y 587.343,Z 367.32,A -85,B 0,C 180,E1 -1428.962,E2 -1428.962} C_VEL
LIN {X 0,Y 587.346,Z 367.325,A -85,B 0,C 180,E1 -1431.744,E2 -1431.744} C_VEL
LIN {X 0,Y 587.362,Z 367.319,A -85,B 0,C 180,E1 -1434.507,E2 -1434.507} C_VEL
LIN {X 0,Y 587.377,Z 367.317,A -85,B 0,C 180,E1 -1437.257,E2 -1437.257} C_VEL
LIN {X 0,Y 587.386,Z 367.321,A -85,B 0,C 180,E1 -1440,E2 -1440} C_VEL
LIN {X 0,Y 587.377,Z 367.315,A -85,B 0,C 180,E1 -1442.743,E2 -1442.743} C_VEL
LIN {X 0,Y 587.361,Z 367.322,A -85,B 0,C 180,E1 -1445.493,E2 -1445.493} C_VEL
LIN {X 0,Y 587.373,Z 367.319,A -85,B 0,C 180,E1 -1448.255,E2 -1448.255} C_VEL
LIN {X 0,Y 587.355,Z 367.319,A -85,B 0,C 180,E1 -1451.134,E2 -1451.134} C_VEL
LIN {X 0,Y 587.372,Z 367.318,A -85,B 0,C 180,E1 -1454.26,E2 -1454.26} C_VEL
LIN {X 0,Y 587.347,Z 367.324,A -85,B 0,C 180,E1 -1457.406,E2 -1457.406} C_VEL
LIN {X 0,Y 587.334,Z 367.324,A -85,B 0,C 180,E1 -1460.305,E2 -1460.305} C_VEL
LIN {X 0,Y 587.319,Z 367.323,A -85,B 0,C 180,E1 -1463.259,E2 -1463.259} C_VEL
LIN {X 0,Y 587.337,Z 367.325,A -85,B 0,C 180,E1 -1465.517,E2 -1465.517} C_VEL
LIN {X 0,Y 587.351,Z 367.322,A -85,B 0,C 180,E1 -1467.818,E2 -1467.818} C_VEL
LIN {X 0,Y 587.342,Z 367.322,A -85,B 0,C 180,E1 -1470.51,E2 -1470.51} C_VEL
LIN {X 0,Y 587.338,Z 367.321,A -85,B 0,C 180,E1 -1473.397,E2 -1473.397} C_VEL
LIN {X 0,Y 587.296,Z 367.332,A -85,B 0,C 180,E1 -1475.9,E2 -1475.9} C_VEL
LIN {X 0,Y 587.335,Z 367.321,A -85,B 0,C 180,E1 -1478.479,E2 -1478.479} C_VEL
LIN {X 0,Y 587.34,Z 367.328,A -85,B 0,C 180,E1 -1481.157,E2 -1481.157} C_VEL
LIN {X 0,Y 587.331,Z 367.323,A -85,B 0,C 180,E1 -1484.113,E2 -1484.113} C_VEL
LIN {X 0,Y 587.326,Z 367.323,A -85,B 0,C 180,E1 -1486.994,E2 -1486.994} C_VEL
LIN {X 0,Y 587.314,Z 367.331,A -85,B 0,C 180,E1 -1489.745,E2 -1489.745} C_VEL
LIN {X 0,Y 587.347,Z 367.321,A -85,B 0,C 180,E1 -1492.392,E2 -1492.392} C_VEL
LIN {X 0,Y 587.349,Z 367.461,A -85,B 0,C 180,E1 -1493.733,E2 -1493.733} C_VEL
LIN {X 0,Y 587.683,Z 372.409,A -85,B 0,C 180,E1 -1495.328,E2 -1495.328} C_VEL
LIN {X 0,Y 587.653,Z 380.45,A -85,B 0,C 180,E1 -1497.82,E2 -1497.82} C_VEL
LIN {X 0,Y 587.569,Z 389.802,A -85,B 0,C 180,E1 -1500.632,E2 -1500.632} C_VEL
LIN {X 0,Y 587.506,Z 399.07,A -85,B 0,C 180,E1 -1503.346,E2 -1503.346} C_VEL
LIN {X 0,Y 587.418,Z 408.337,A -85,B 0,C 180,E1 -1505.997,E2 -1505.997} C_VEL
LIN {X 0,Y 587.357,Z 417.606,A -85,B 0,C 180,E1 -1508.596,E2 -1508.596} C_VEL
LIN {X 0,Y 587.324,Z 428.196,A -85,B 0,C 180,E1 -1511.512,E2 -1511.512} C_VEL
LIN {X 0,Y 587.262,Z 438.787,A -85,B 0,C 180,E1 -1514.379,E2 -1514.379} C_VEL
LIN {X 0,Y 587.25,Z 449.378,A -85,B 0,C 180,E1 -1517.208,E2 -1517.208} C_VEL
LIN {X 0,Y 587.216,Z 451.571,A -85,B 0,C 180,E1 -1517.789,E2 -1517.789} C_VEL
LIN {X 0,Y 587.735,Z 457.222,A -85,B 0,C 180,E1 -1517.899,E2 -1517.899} C_VEL
LIN {X 0,Y 587.687,Z 470.491,A -85,B 0,C 180,E1 -1518.226,E2 -1518.226} C_VEL
LIN {X 0,Y 587.622,Z 482.227,A -85,B 0,C 180,E1 -1518.649,E2 -1518.649} C_VEL
LIN {X 0,Y 587.544,Z 494.206,A -85,B 0,C 180,E1 -1519.228,E2 -1519.228} C_VEL
LIN {X 0,Y 587.463,Z 505.474,A -85,B 0,C 180,E1 -1519.923,E2 -1519.923} C_VEL
LIN {X 0,Y 587.384,Z 515.645,A -85,B 0,C 180,E1 -1520.704,E2 -1520.704} C_VEL
LIN {X 0,Y 587.34,Z 524.786,A -85,B 0,C 180,E1 -1521.571,E2 -1521.571} C_VEL
LIN {X 0,Y 587.259,Z 533.69,A -85,B 0,C 180,E1 -1522.608,E2 -1522.608} C_VEL
LIN {X 0,Y 587.195,Z 540.745,A -85,B 0,C 180,E1 -1523.627,E2 -1523.627} C_VEL
LIN {X 0,Y 587.211,Z 545.68,A -85,B 0,C 180,E1 -1524.506,E2 -1524.506} C_VEL
LIN {X 0,Y 587.188,Z 550.371,A -85,B 0,C 180,E1 -1525.538,E2 -1525.538} C_VEL
LIN {X 0,Y 587.193,Z 553.956,A -85,B 0,C 180,E1 -1526.569,E2 -1526.569} C_VEL
LIN {X 0,Y 587.132,Z 555.809,A -85,B 0,C 180,E1 -1527.256,E2 -1527.256} C_VEL
LIN {X 0,Y 587.141,Z 557.202,A -85,B 0,C 180,E1 -1527.942,E2 -1527.942} C_VEL
LIN {X 0,Y 587.14,Z 558.784,A -85,B 0,C 180,E1 -1529.314,E2 -1529.314} C_VEL
LIN {X 0,Y 587.137,Z 559,A -85,B 0,C 180,E1 -1530,E2 -1530} C_VEL
LIN {X 0,Y 587.147,Z 558.185,A -85,B 0,C 180,E1 -1531.372,E2 -1531.372} C_VEL
LIN {X 0,Y 587.141,Z 557.202,A -85,B 0,C 180,E1 -1532.058,E2 -1532.058} C_VEL
LIN {X 0,Y 587.132,Z 555.81,A -85,B 0,C 180,E1 -1532.744,E2 -1532.744} C_VEL
LIN {X 0,Y 587.212,Z 552.896,A -85,B 0,C 180,E1 -1533.774,E2 -1533.774} C_VEL
LIN {X 0,Y 587.147,Z 548.95,A -85,B 0,C 180,E1 -1534.806,E2 -1534.806} C_VEL
LIN {X 0,Y 587.217,Z 542.877,A -85,B 0,C 180,E1 -1536.011,E2 -1536.011} C_VEL
LIN {X 0,Y 587.245,Z 536.236,A -85,B 0,C 180,E1 -1537.046,E2 -1537.046} C_VEL
LIN {X 0,Y 587.299,Z 527.99,A -85,B 0,C 180,E1 -1538.083,E2 -1538.083} C_VEL
LIN {X 0,Y 587.343,Z 519.537,A -85,B 0,C 180,E1 -1538.949,E2 -1538.949} C_VEL
LIN {X 0,Y 587.422,Z 509.093,A -85,B 0,C 180,E1 -1539.816,E2 -1539.816} C_VEL
LIN {X 0,Y 587.486,Z 498.758,A -85,B 0,C 180,E1 -1540.512,E2 -1540.512} C_VEL
LIN {X 0,Y 587.561,Z 486.814,A -85,B 0,C 180,E1 -1541.149,E2 -1541.149} C_VEL
LIN {X 0,Y 587.635,Z 474.598,A -85,B 0,C 180,E1 -1541.639,E2 -1541.639} C_VEL
LIN {X 0,Y 587.72,Z 461.437,A -85,B 0,C 180,E1 -1542.014,E2 -1542.014} C_VEL
LIN {X 0,Y 587.505,Z 453.612,A -85,B 0,C 180,E1 -1542.171,E2 -1542.171} C_VEL
LIN {X 0,Y 587.215,Z 451.53,A -85,B 0,C 180,E1 -1542.221,E2 -1542.221} C_VEL
LIN {X 0,Y 587.27,Z 441.435,A -85,B 0,C 180,E1 -1544.91,E2 -1544.91} C_VEL
LIN {X 0,Y 587.302,Z 430.844,A -85,B 0,C 180,E1 -1547.767,E2 -1547.767} C_VEL
LIN {X 0,Y 587.378,Z 420.253,A -85,B 0,C 180,E1 -1550.669,E2 -1550.669} C_VEL
LIN {X 0,Y 587.433,Z 409.662,A -85,B 0,C 180,E1 -1553.628,E2 -1553.628} C_VEL
LIN {X 0,Y 587.495,Z 400.394,A -85,B 0,C 180,E1 -1556.271,E2 -1556.271} C_VEL
LIN {X 0,Y 587.513,Z 392.451,A -85,B 0,C 180,E1 -1558.587,E2 -1558.587} C_VEL
LIN {X 0,Y 587.62,Z 383.183,A -85,B 0,C 180,E1 -1561.35,E2 -1561.35} C_VEL
LIN {X 0,Y 587.665,Z 373.916,A -85,B 0,C 180,E1 -1564.2,E2 -1564.2} C_VEL
LIN {X 0,Y 587.557,Z 368.62,A -85,B 0,C 180,E1 -1565.881,E2 -1565.881} C_VEL
LIN {X 0,Y 587.316,Z 367.33,A -85,B 0,C 180,E1 -1566.323,E2 -1566.323} C_VEL
LIN {X 0,Y 587.324,Z 367.326,A -85,B 0,C 180,E1 -1568.94,E2 -1568.94} C_VEL
LIN {X 0,Y 587.357,Z 367.326,A -85,B 0,C 180,E1 -1572.072,E2 -1572.072} C_VEL
LIN {X 0,Y 587.32,Z 367.327,A -85,B 0,C 180,E1 -1575.089,E2 -1575.089} C_VEL
LIN {X 0,Y 587.326,Z 367.322,A -85,B 0,C 180,E1 -1577.925,E2 -1577.925} C_VEL
LIN {X 0,Y 587.349,Z 367.326,A -85,B 0,C 180,E1 -1580.641,E2 -1580.641} C_VEL
LIN {X 0,Y 587.353,Z 367.319,A -85,B 0,C 180,E1 -1583.292,E2 -1583.292} C_VEL
LIN {X 0,Y 587.366,Z 367.324,A -85,B 0,C 180,E1 -1585.78,E2 -1585.78} C_VEL
LIN {X 0,Y 587.345,Z 367.32,A -85,B 0,C 180,E1 -1588.231,E2 -1588.231} C_VEL
LIN {X 0,Y 587.352,Z 367.326,A -85,B 0,C 180,E1 -1590.867,E2 -1590.867} C_VEL
LIN {X 0,Y 587.363,Z 367.319,A -85,B 0,C 180,E1 -1593.819,E2 -1593.819} C_VEL
LIN {X 0,Y 587.334,Z 367.328,A -85,B 0,C 180,E1 -1595.993,E2 -1595.993} C_VEL
LIN {X 0,Y 587.325,Z 367.323,A -85,B 0,C 180,E1 -1598.226,E2 -1598.226} C_VEL
LIN {X 0,Y 587.354,Z 367.325,A -85,B 0,C 180,E1 -1601.151,E2 -1601.151} C_VEL
LIN {X 0,Y 587.328,Z 367.323,A -85,B 0,C 180,E1 -1604.025,E2 -1604.025} C_VEL
LIN {X 0,Y 587.366,Z 367.323,A -85,B 0,C 180,E1 -1606.154,E2 -1606.154} C_VEL
LIN {X 0,Y 587.343,Z 367.32,A -85,B 0,C 180,E1 -1608.962,E2 -1608.962} C_VEL
LIN {X 0,Y 587.373,Z 367.319,A -85,B 0,C 180,E1 -1611.745,E2 -1611.745} C_VEL
LIN {X 0,Y 587.36,Z 367.322,A -85,B 0,C 180,E1 -1614.507,E2 -1614.507} C_VEL
LIN {X 0,Y 587.377,Z 367.315,A -85,B 0,C 180,E1 -1617.257,E2 -1617.257} C_VEL
LIN {X 0,Y 587.385,Z 367.322,A -85,B 0,C 180,E1 -1620,E2 -1620} C_VEL
LIN {X 0,Y 587.377,Z 367.317,A -85,B 0,C 180,E1 -1622.743,E2 -1622.743} C_VEL
LIN {X 0,Y 587.362,Z 367.32,A -85,B 0,C 180,E1 -1625.493,E2 -1625.493} C_VEL
LIN {X 0,Y 587.346,Z 367.324,A -85,B 0,C 180,E1 -1628.256,E2 -1628.256} C_VEL
LIN {X 0,Y 587.353,Z 367.318,A -85,B 0,C 180,E1 -1631.134,E2 -1631.134} C_VEL
LIN {X 0,Y 587.369,Z 367.317,A -85,B 0,C 180,E1 -1634.26,E2 -1634.26} C_VEL
LIN {X 0,Y 587.349,Z 367.322,A -85,B 0,C 180,E1 -1637.406,E2 -1637.406} C_VEL
LIN {X 0,Y 587.307,Z 367.326,A -85,B 0,C 180,E1 -1638.312,E2 -1638.312} C_VEL
LIN {X 0,Y 586.667,Z 367.41,A -85,B 0,C 180,E1 -1638.885,E2 -1638.885} C_VEL
LIN {X 0,Y 583.845,Z 367.758,A -85,B 0,C 180,E1 -1639.813,E2 -1639.813} C_VEL
LIN {X 0,Y 581.436,Z 368.062,A -85,B 0,C 180,E1 -1640.56,E2 -1640.56} C_VEL
LIN {X 0,Y 580.382,Z 368.188,A -85,B 0,C 180,E1 -1641.137,E2 -1641.137} C_VEL
LIN {X 0,Y 580.287,Z 368.199,A -85,B 0,C 180,E1 -1641.332,E2 -1641.332} C_VEL
LIN {X 0,Y 580.303,Z 368.199,A -85,B 0,C 180,E1 -1644.316,E2 -1644.316} C_VEL
LIN {X 0,Y 580.281,Z 368.2,A -85,B 0,C 180,E1 -1646.623,E2 -1646.623} C_VEL
LIN {X 0,Y 580.305,Z 368.201,A -85,B 0,C 180,E1 -1649.31,E2 -1649.31} C_VEL
LIN {X 0,Y 580.302,Z 368.201,A -85,B 0,C 180,E1 -1652.2,E2 -1652.2} C_VEL
LIN {X 0,Y 580.295,Z 368.199,A -85,B 0,C 180,E1 -1654.696,E2 -1654.696} C_VEL
LIN {X 0,Y 580.302,Z 368.2,A -85,B 0,C 180,E1 -1657.268,E2 -1657.268} C_VEL
LIN {X 0,Y 580.3,Z 368.198,A -85,B 0,C 180,E1 -1660.271,E2 -1660.271} C_VEL
LIN {X 0,Y 580.28,Z 368.207,A -85,B 0,C 180,E1 -1662.706,E2 -1662.706} C_VEL
LIN {X 0,Y 580.276,Z 368.202,A -85,B 0,C 180,E1 -1665.609,E2 -1665.609} C_VEL
LIN {X 0,Y 580.318,Z 368.197,A -85,B 0,C 180,E1 -1668.234,E2 -1668.234} C_VEL
LIN {X 0,Y 580.282,Z 368.203,A -85,B 0,C 180,E1 -1670.965,E2 -1670.965} C_VEL
LIN {X 0,Y 580.267,Z 368.202,A -85,B 0,C 180,E1 -1673.596,E2 -1673.596} C_VEL
LIN {X 0,Y 580.185,Z 368.385,A -85,B 0,C 180,E1 -1675.458,E2 -1675.458} C_VEL
LIN {X 0,Y 580.164,Z 371.149,A -85,B 0,C 180,E1 -1677.992,E2 -1677.992} C_VEL
LIN {X 0,Y 580.158,Z 374.156,A -85,B 0,C 180,E1 -1680.716,E2 -1680.716} C_VEL
LIN {X 0,Y 580.129,Z 377.534,A -85,B 0,C 180,E1 -1683.699,E2 -1683.699} C_VEL
LIN {X 0,Y 580.068,Z 380.806,A -85,B 0,C 180,E1 -1686.433,E2 -1686.433} C_VEL
LIN {X 0,Y 580.086,Z 384.65,A -85,B 0,C 180,E1 -1689.43,E2 -1689.43} C_VEL
LIN {X 0,Y 580.043,Z 388.493,A -85,B 0,C 180,E1 -1692.368,E2 -1692.368} C_VEL
LIN {X 0,Y 580.054,Z 391.375,A -85,B 0,C 180,E1 -1694.541,E2 -1694.541} C_VEL
LIN {X 0,Y 580.06,Z 394.258,A -85,B 0,C 180,E1 -1696.691,E2 -1696.691} C_VEL
LIN {X 0,Y 580.077,Z 395.669,A -85,B 0,C 180,E1 -1697.737,E2 -1697.737} C_VEL
LIN {X 0,Y 580.777,Z 401.406,A -85,B 0,C 180,E1 -1697.885,E2 -1697.885} C_VEL
LIN {X 0,Y 580.666,Z 414.451,A -85,B 0,C 180,E1 -1698.259,E2 -1698.259} C_VEL
LIN {X 0,Y 580.596,Z 426.325,A -85,B 0,C 180,E1 -1698.739,E2 -1698.739} C_VEL
LIN {X 0,Y 580.51,Z 438.03,A -85,B 0,C 180,E1 -1699.361,E2 -1699.361} C_VEL
LIN {X 0,Y 580.396,Z 449.664,A -85,B 0,C 180,E1 -1700.152,E2 -1700.152} C_VEL
LIN {X 0,Y 580.308,Z 459.044,A -85,B 0,C 180,E1 -1700.942,E2 -1700.942} C_VEL
LIN {X 0,Y 580.251,Z 467.605,A -85,B 0,C 180,E1 -1701.818,E2 -1701.818} C_VEL
LIN {X 0,Y 580.205,Z 475.919,A -85,B 0,C 180,E1 -1702.868,E2 -1702.868} C_VEL
LIN {X 0,Y 580.14,Z 482.618,A -85,B 0,C 180,E1 -1703.915,E2 -1703.915} C_VEL
LIN {X 0,Y 580.053,Z 488.76,A -85,B 0,C 180,E1 -1705.135,E2 -1705.135} C_VEL
LIN {X 0,Y 580.11,Z 492.75,A -85,B 0,C 180,E1 -1706.179,E2 -1706.179} C_VEL
LIN {X 0,Y 580.043,Z 495.698,A -85,B 0,C 180,E1 -1707.222,E2 -1707.222} C_VEL
LIN {X 0,Y 580.04,Z 497.128,A -85,B 0,C 180,E1 -1707.917,E2 -1707.917} C_VEL
LIN {X 0,Y 580.04,Z 498.755,A -85,B 0,C 180,E1 -1709.306,E2 -1709.306} C_VEL
LIN {X 0,Y 580.038,Z 498.996,A -85,B 0,C 180,E1 -1710,E2 -1710} C_VEL
LIN {X 0,Y 580.04,Z 498.815,A -85,B 0,C 180,E1 -1710.694,E2 -1710.694} C_VEL
LIN {X 0,Y 580.04,Z 497.272,A -85,B 0,C 180,E1 -1712.083,E2 -1712.083} C_VEL
LIN {X 0,Y 580.044,Z 495.911,A -85,B 0,C 180,E1 -1712.778,E2 -1712.778} C_VEL
LIN {X 0,Y 580.11,Z 493.034,A -85,B 0,C 180,E1 -1713.821,E2 -1713.821} C_VEL
LIN {X 0,Y 580.053,Z 489.133,A -85,B 0,C 180,E1 -1714.865,E2 -1714.865} C_VEL
LIN {X 0,Y 580.162,Z 484.101,A -85,B 0,C 180,E1 -1715.91,E2 -1715.91} C_VEL
LIN {X 0,Y 580.158,Z 477.779,A -85,B 0,C 180,E1 -1716.958,E2 -1716.958} C_VEL
LIN {X 0,Y 580.241,Z 469.859,A -85,B 0,C 180,E1 -1718.007,E2 -1718.007} C_VEL
LIN {X 0,Y 580.308,Z 460.01,A -85,B 0,C 180,E1 -1719.058,E2 -1719.058} C_VEL
LIN {X 0,Y 580.421,Z 449.688,A -85,B 0,C 180,E1 -1719.936,E2 -1719.936} C_VEL
LIN {X 0,Y 580.524,Z 438.055,A -85,B 0,C 180,E1 -1720.727,E2 -1720.727} C_VEL
LIN {X 0,Y 580.619,Z 426.417,A -85,B 0,C 180,E1 -1721.347,E2 -1721.347} C_VEL
LIN {X 0,Y 580.668,Z 414.619,A -85,B 0,C 180,E1 -1721.825,E2 -1721.825} C_VEL
LIN {X 0,Y 580.781,Z 401.459,A -85,B 0,C 180,E1 -1722.204,E2 -1722.204} C_VEL
LIN {X 0,Y 580.091,Z 395.671,A -85,B 0,C 180,E1 -1722.352,E2 -1722.352} C_VEL
LIN {X 0,Y 580.045,Z 392.457,A -85,B 0,C 180,E1 -1724.741,E2 -1724.741} C_VEL
LIN {X 0,Y 580.067,Z 389.573,A -85,B 0,C 180,E1 -1726.905,E2 -1726.905} C_VEL
LIN {X 0,Y 580.065,Z 385.727,A -85,B 0,C 180,E1 -1729.831,E2 -1729.831} C_VEL
LIN {X 0,Y 580.047,Z 382.843,A -85,B 0,C 180,E1 -1732.062,E2 -1732.062} C_VEL
LIN {X 0,Y 580.097,Z 379.511,A -85,B 0,C 180,E1 -1734.681,E2 -1734.681} C_VEL
LIN {X 0,Y 580.122,Z 376.366,A -85,B 0,C 180,E1 -1737.411,E2 -1737.411} C_VEL
LIN {X 0,Y 580.144,Z 373.688,A -85,B 0,C 180,E1 -1739.781,E2 -1739.781} C_VEL
LIN {X 0,Y 580.152,Z 371.026,A -85,B 0,C 180,E1 -1742.21,E2 -1742.21} C_VEL
LIN {X 0,Y 580.181,Z 368.306,A -85,B 0,C 180,E1 -1744.704,E2 -1744.704} C_VEL
LIN {X 0,Y 580.303,Z 368.202,A -85,B 0,C 180,E1 -1747.269,E2 -1747.269} C_VEL
LIN {X 0,Y 580.296,Z 368.202,A -85,B 0,C 180,E1 -1750.271,E2 -1750.271} C_VEL
LIN {X 0,Y 580.286,Z 368.201,A -85,B 0,C 180,E1 -1752.706,E2 -1752.706} C_VEL
LIN {X 0,Y 580.262,Z 368.209,A -85,B 0,C 180,E1 -1755.61,E2 -1755.61} C_VEL
LIN {X 0,Y 580.283,Z 368.2,A -85,B 0,C 180,E1 -1758.231,E2 -1758.231} C_VEL
LIN {X 0,Y 580.295,Z 368.203,A -85,B 0,C 180,E1 -1760.966,E2 -1760.966} C_VEL
LIN {X 0,Y 580.274,Z 368.201,A -85,B 0,C 180,E1 -1763.597,E2 -1763.597} C_VEL
LIN {X 0,Y 580.323,Z 368.199,A -85,B 0,C 180,E1 -1766.146,E2 -1766.146} C_VEL
LIN {X 0,Y 580.281,Z 368.2,A -85,B 0,C 180,E1 -1768.615,E2 -1768.615} C_VEL
LIN {X 0,Y 580.296,Z 368.205,A -85,B 0,C 180,E1 -1771.024,E2 -1771.024} C_VEL
LIN {X 0,Y 580.295,Z 368.198,A -85,B 0,C 180,E1 -1773.666,E2 -1773.666} C_VEL
LIN {X 0,Y 580.304,Z 368.198,A -85,B 0,C 180,E1 -1775.684,E2 -1775.684} C_VEL
LIN {X 0,Y 580.29,Z 368.198,A -85,B 0,C 180,E1 -1778.695,E2 -1778.695} C_VEL
LIN {X 0,Y 580.307,Z 368.199,A -85,B 0,C 180,E1 -1780.914,E2 -1780.914} C_VEL
LIN {X 0,Y 580.274,Z 368.201,A -85,B 0,C 180,E1 -1783.825,E2 -1783.825} C_VEL
LIN {X 0,Y 580.331,Z 368.196,A -85,B 0,C 180,E1 -1785.983,E2 -1785.983} C_VEL
LIN {X 0,Y 580.311,Z 368.196,A -85,B 0,C 180,E1 -1788.827,E2 -1788.827} C_VEL
LIN {X 0,Y 580.316,Z 368.202,A -85,B 0,C 180,E1 -1791.644,E2 -1791.644} C_VEL
LIN {X 0,Y 580.284,Z 368.201,A -85,B 0,C 180,E1 -1793.742,E2 -1793.742} C_VEL
LIN {X 0,Y 580.267,Z 368.202,A -85,B 0,C 180,E1 -1795.833,E2 -1795.833} C_VEL
LIN {X 0,Y 580.336,Z 368.195,A -85,B 0,C 180,E1 -1797.918,E2 -1797.918} C_VEL
LIN {X 0,Y 580.365,Z 368.19,A -85,B 0,C 180,E1 -1800.694,E2 -1800.694} C_VEL
LIN {X 0,Y 580.284,Z 368.206,A -85,B 0,C 180,E1 -1803.472,E2 -1803.472} C_VEL
LIN {X 0,Y 580.327,Z 368.197,A -85,B 0,C 180,E1 -1805.56,E2 -1805.56} C_VEL
LIN {X 0,Y 580.338,Z 368.196,A -85,B 0,C 180,E1 -1808.356,E2 -1808.356} C_VEL
LIN {X 0,Y 580.306,Z 368.197,A -85,B 0,C 180,E1 -1811.191,E2 -1811.191} C_VEL
LIN {X 0,Y 580.333,Z 368.197,A -85,B 0,C 180,E1 -1814.017,E2 -1814.017} C_VEL
LIN {X 0,Y 580.318,Z 368.198,A -85,B 0,C 180,E1 -1816.914,E2 -1816.914} C_VEL
LIN {X 0,Y 580.31,Z 368.196,A -85,B 0,C 180,E1 -1819.822,E2 -1819.822} C_VEL
LIN {X 0,Y 580.295,Z 368.2,A -85,B 0,C 180,E1 -1822.802,E2 -1822.802} C_VEL
LIN {X 0,Y 580.311,Z 368.196,A -85,B 0,C 180,E1 -1825.08,E2 -1825.08} C_VEL
LIN {X 0,Y 580.303,Z 368.197,A -85,B 0,C 180,E1 -1828.185,E2 -1828.185} C_VEL
LIN {X 0,Y 580.289,Z 368.203,A -85,B 0,C 180,E1 -1830.694,E2 -1830.694} C_VEL
LIN {X 0,Y 580.307,Z 368.197,A -85,B 0,C 180,E1 -1833.316,E2 -1833.316} C_VEL
LIN {X 0,Y 580.251,Z 368.207,A -85,B 0,C 180,E1 -1835.756,E2 -1835.756} C_VEL
LIN {X 0,Y 580.292,Z 368.201,A -85,B 0,C 180,E1 -1838.146,E2 -1838.146} C_VEL
LIN {X 0,Y 580.303,Z 368.2,A -85,B 0,C 180,E1 -1840.843,E2 -1840.843} C_VEL
LIN {X 0,Y 580.283,Z 368.2,A -85,B 0,C 180,E1 -1843.658,E2 -1843.658} C_VEL
LIN {X 0,Y 580.29,Z 368.202,A -85,B 0,C 180,E1 -1846.608,E2 -1846.608} C_VEL
LIN {X 0,Y 580.301,Z 368.199,A -85,B 0,C 180,E1 -1849.156,E2 -1849.156} C_VEL
LIN {X 0,Y 580.293,Z 368.202,A -85,B 0,C 180,E1 -1851.927,E2 -1851.927} C_VEL
LIN {X 0,Y 580.321,Z 368.328,A -85,B 0,C 180,E1 -1853.505,E2 -1853.505} C_VEL
LIN {X 0,Y 580.744,Z 372.592,A -85,B 0,C 180,E1 -1854.912,E2 -1854.912} C_VEL
LIN {X 0,Y 580.702,Z 381.859,A -85,B 0,C 180,E1 -1857.824,E2 -1857.824} C_VEL
LIN {X 0,Y 580.568,Z 391.135,A -85,B 0,C 180,E1 -1860.644,E2 -1860.644} C_VEL
LIN {X 0,Y 580.499,Z 400.394,A -85,B 0,C 180,E1 -1863.387,E2 -1863.387} C_VEL
LIN {X 0,Y 580.421,Z 409.661,A -85,B 0,C 180,E1 -1866.069,E2 -1866.069} C_VEL
LIN {X 0,Y 580.323,Z 419.404,A -85,B 0,C 180,E1 -1868.83,E2 -1868.83} C_VEL
LIN {X 0,Y 580.26,Z 428.196,A -85,B 0,C 180,E1 -1871.279,E2 -1871.279} C_VEL
LIN {X 0,Y 580.222,Z 437.463,A -85,B 0,C 180,E1 -1873.824,E2 -1873.824} C_VEL
LIN {X 0,Y 580.19,Z 448.054,A -85,B 0,C 180,E1 -1876.694,E2 -1876.694} C_VEL
LIN {X 0,Y 580.151,Z 451.53,A -85,B 0,C 180,E1 -1877.627,E2 -1877.627} C_VEL
LIN {X 0,Y 580.815,Z 457.222,A -85,B 0,C 180,E1 -1877.753,E2 -1877.753} C_VEL
LIN {X 0,Y 580.728,Z 469.731,A -85,B 0,C 180,E1 -1878.061,E2 -1878.061} C_VEL
LIN {X 0,Y 580.654,Z 482.524,A -85,B 0,C 180,E1 -1878.524,E2 -1878.524} C_VEL
LIN {X 0,Y 580.562,Z 494.206,A -85,B 0,C 180,E1 -1879.097,E2 -1879.097} C_VEL
LIN {X 0,Y 580.452,Z 505.475,A -85,B 0,C 180,E1 -1879.8,E2 -1879.8} C_VEL
LIN {X 0,Y 580.352,Z 515.645,A -85,B 0,C 180,E1 -1880.591,E2 -1880.591} C_VEL
LIN {X 0,Y 580.279,Z 524.786,A -85,B 0,C 180,E1 -1881.468,E2 -1881.468} C_VEL
LIN {X 0,Y 580.199,Z 533.69,A -85,B 0,C 180,E1 -1882.518,E2 -1882.518} C_VEL
LIN {X 0,Y 580.12,Z 540.465,A -85,B 0,C 180,E1 -1883.505,E2 -1883.505} C_VEL
LIN {X 0,Y 580.139,Z 545.68,A -85,B 0,C 180,E1 -1884.438,E2 -1884.438} C_VEL
LIN {X 0,Y 580.108,Z 550.371,A -85,B 0,C 180,E1 -1885.483,E2 -1885.483} C_VEL
LIN {X 0,Y 580.123,Z 553.956,A -85,B 0,C 180,E1 -1886.527,E2 -1886.527} C_VEL
LIN {X 0,Y 580.043,Z 555.809,A -85,B 0,C 180,E1 -1887.222,E2 -1887.222} C_VEL
LIN {X 0,Y 580.04,Z 557.201,A -85,B 0,C 180,E1 -1887.917,E2 -1887.917} C_VEL
LIN {X 0,Y 580.04,Z 558.784,A -85,B 0,C 180,E1 -1889.306,E2 -1889.306} C_VEL
LIN {X 0,Y 580.037,Z 559,A -85,B 0,C 180,E1 -1890,E2 -1890} C_VEL
LIN {X 0,Y 580.047,Z 558.185,A -85,B 0,C 180,E1 -1891.388,E2 -1891.388} C_VEL
LIN {X 0,Y 580.04,Z 557.202,A -85,B 0,C 180,E1 -1892.083,E2 -1892.083} C_VEL
LIN {X 0,Y 580.043,Z 555.81,A -85,B 0,C 180,E1 -1892.778,E2 -1892.778} C_VEL
LIN {X 0,Y 580.109,Z 552.896,A -85,B 0,C 180,E1 -1893.821,E2 -1893.821} C_VEL
LIN {X 0,Y 580.054,Z 548.95,A -85,B 0,C 180,E1 -1894.865,E2 -1894.865} C_VEL
LIN {X 0,Y 580.139,Z 542.878,A -85,B 0,C 180,E1 -1896.085,E2 -1896.085} C_VEL
LIN {X 0,Y 580.184,Z 536.236,A -85,B 0,C 180,E1 -1897.132,E2 -1897.132} C_VEL
LIN {X 0,Y 580.25,Z 527.99,A -85,B 0,C 180,E1 -1898.182,E2 -1898.182} C_VEL
LIN {X 0,Y 580.308,Z 519.537,A -85,B 0,C 180,E1 -1899.058,E2 -1899.058} C_VEL
LIN {X 0,Y 580.425,Z 509.093,A -85,B 0,C 180,E1 -1899.936,E2 -1899.936} C_VEL
LIN {X 0,Y 580.491,Z 498.758,A -85,B 0,C 180,E1 -1900.64,E2 -1900.64} C_VEL
LIN {X 0,Y 580.596,Z 487.247,A -85,B 0,C 180,E1 -1901.264,E2 -1901.264} C_VEL
LIN {X 0,Y 580.677,Z 474.471,A -85,B 0,C 180,E1 -1901.785,E2 -1901.785} C_VEL
LIN {X 0,Y 580.785,Z 461.436,A -85,B 0,C 180,E1 -1902.159,E2 -1902.159} C_VEL
LIN {X 0,Y 580.551,Z 454.162,A -85,B 0,C 180,E1 -1902.311,E2 -1902.311} C_VEL
LIN {X 0,Y 580.151,Z 451.53,A -85,B 0,C 180,E1 -1902.373,E2 -1902.373} C_VEL
LIN {X 0,Y 580.227,Z 441.435,A -85,B 0,C 180,E1 -1905.095,E2 -1905.095} C_VEL
LIN {X 0,Y 580.253,Z 430.844,A -85,B 0,C 180,E1 -1907.99,E2 -1907.99} C_VEL
LIN {X 0,Y 580.345,Z 420.491,A -85,B 0,C 180,E1 -1910.865,E2 -1910.865} C_VEL
LIN {X 0,Y 580.405,Z 410.985,A -85,B 0,C 180,E1 -1913.553,E2 -1913.553} C_VEL
LIN {X 0,Y 580.452,Z 403.042,A -85,B 0,C 180,E1 -1915.841,E2 -1915.841} C_VEL
LIN {X 0,Y 580.536,Z 393.775,A -85,B 0,C 180,E1 -1918.567,E2 -1918.567} C_VEL
LIN {X 0,Y 580.639,Z 384.507,A -85,B 0,C 180,E1 -1921.364,E2 -1921.364} C_VEL
LIN {X 0,Y 580.731,Z 375.315,A -85,B 0,C 180,E1 -1924.222,E2 -1924.222} C_VEL
LIN {X 0,Y 580.648,Z 370.364,A -85,B 0,C 180,E1 -1925.811,E2 -1925.811} C_VEL
LIN {X 0,Y 580.307,Z 368.204,A -85,B 0,C 180,E1 -1926.591,E2 -1926.591} C_VEL
LIN {X 0,Y 580.297,Z 368.2,A -85,B 0,C 180,E1 -1929.185,E2 -1929.185} C_VEL
LIN {X 0,Y 580.318,Z 368.2,A -85,B 0,C 180,E1 -1931.766,E2 -1931.766} C_VEL
LIN {X 0,Y 580.273,Z 368.202,A -85,B 0,C 180,E1 -1934.626,E2 -1934.626} C_VEL
LIN {X 0,Y 580.289,Z 368.2,A -85,B 0,C 180,E1 -1937.628,E2 -1937.628} C_VEL
LIN {X 0,Y 580.297,Z 368.199,A -85,B 0,C 180,E1 -1940.067,E2 -1940.067} C_VEL
LIN {X 0,Y 580.303,Z 368.197,A -85,B 0,C 180,E1 -1943.066,E2 -1943.066} C_VEL
LIN {X 0,Y 580.32,Z 368.197,A -85,B 0,C 180,E1 -1946.145,E2 -1946.145} C_VEL
LIN {X 0,Y 580.28,Z 368.201,A -85,B 0,C 180,E1 -1948.615,E2 -1948.615} C_VEL
LIN {X 0,Y 580.295,Z 368.202,A -85,B 0,C 180,E1 -1951.024,E2 -1951.024} C_VEL
LIN {X 0,Y 580.296,Z 368.199,A -85,B 0,C 180,E1 -1953.666,E2 -1953.666} C_VEL
LIN {X 0,Y 580.303,Z 368.201,A -85,B 0,C 180,E1 -1955.684,E2 -1955.684} C_VEL
LIN {X 0,Y 580.289,Z 368.199,A -85,B 0,C 180,E1 -1958.695,E2 -1958.695} C_VEL
LIN {X 0,Y 580.324,Z 368.199,A -85,B 0,C 180,E1 -1960.914,E2 -1960.914} C_VEL
LIN {X 0,Y 580.281,Z 368.199,A -85,B 0,C 180,E1 -1963.826,E2 -1963.826} C_VEL
LIN {X 0,Y 580.332,Z 368.197,A -85,B 0,C 180,E1 -1965.983,E2 -1965.983} C_VEL
LIN {X 0,Y 580.31,Z 368.196,A -85,B 0,C 180,E1 -1968.827,E2 -1968.827} C_VEL
LIN {X 0,Y 580.337,Z 368.197,A -85,B 0,C 180,E1 -1971.644,E2 -1971.644} C_VEL
LIN {X 0,Y 580.326,Z 368.197,A -85,B 0,C 180,E1 -1974.44,E2 -1974.44} C_VEL
LIN {X 0,Y 580.343,Z 368.192,A -85,B 0,C 180,E1 -1977.224,E2 -1977.224} C_VEL
LIN {X 0,Y 580.355,Z 368.197,A -85,B 0,C 180,E1 -1980,E2 -1980} C_VEL
LIN {X 0,Y 580.343,Z 368.193,A -85,B 0,C 180,E1 -1982.777,E2 -1982.777} C_VEL
LIN {X 0,Y 580.327,Z 368.196,A -85,B 0,C 180,E1 -1985.56,E2 -1985.56} C_VEL
LIN {X 0,Y 580.328,Z 368.194,A -85,B 0,C 180,E1 -1987.655,E2 -1987.655} C_VEL
LIN {X 0,Y 580.302,Z 368.201,A -85,B 0,C 180,E1 -1990.467,E2 -1990.467} C_VEL
LIN {X 0,Y 580.308,Z 368.197,A -85,B 0,C 180,E1 -1992.591,E2 -1992.591} C_VEL
LIN {X 0,Y 580.29,Z 368.199,A -85,B 0,C 180,E1 -1994.734,E2 -1994.734} C_VEL
LIN {X 0,Y 580.292,Z 368.199,A -85,B 0,C 180,E1 -1997.625,E2 -1997.625} C_VEL
LIN {X 0,Y 580.31,Z 368.197,A -85,B 0,C 180,E1 -1999.822,E2 -1999.822} C_VEL
LIN {X 0,Y 580.287,Z 368.199,A -85,B 0,C 180,E1 -2001.332,E2 -2001.332} C_VEL
LIN {X 0,Y 579.59,Z 368.291,A -85,B 0,C 180,E1 -2001.911,E2 -2001.911} C_VEL
LIN {X 0,Y 576.712,Z 368.648,A -85,B 0,C 180,E1 -2002.851,E2 -2002.851} C_VEL
LIN {X 0,Y 574.317,Z 368.946,A -85,B 0,C 180,E1 -2003.607,E2 -2003.607} C_VEL
LIN {X 0,Y 573.319,Z 369.07,A -85,B 0,C 180,E1 -2004.191,E2 -2004.191} C_VEL
LIN {X 0,Y 573.254,Z 369.076,A -85,B 0,C 180,E1 -2004.389,E2 -2004.389} C_VEL
LIN {X 0,Y 573.255,Z 369.078,A -85,B 0,C 180,E1 -2006.976,E2 -2006.976} C_VEL
LIN {X 0,Y 573.25,Z 369.078,A -85,B 0,C 180,E1 -2009.488,E2 -2009.488} C_VEL
LIN {X 0,Y 573.258,Z 369.079,A -85,B 0,C 180,E1 -2012.645,E2 -2012.645} C_VEL
LIN {X 0,Y 573.212,Z 369.08,A -85,B 0,C 180,E1 -2015.188,E2 -2015.188} C_VEL
LIN {X 0,Y 573.24,Z 369.081,A -85,B 0,C 180,E1 -2017.807,E2 -2017.807} C_VEL
LIN {X 0,Y 573.274,Z 369.074,A -85,B 0,C 180,E1 -2020.528,E2 -2020.528} C_VEL
LIN {X 0,Y 573.242,Z 369.077,A -85,B 0,C 180,E1 -2023.668,E2 -2023.668} C_VEL
LIN {X 0,Y 573.251,Z 369.077,A -85,B 0,C 180,E1 -2026.642,E2 -2026.642} C_VEL
LIN {X 0,Y 573.248,Z 369.082,A -85,B 0,C 180,E1 -2029.475,E2 -2029.475} C_VEL
LIN {X 0,Y 573.239,Z 369.077,A -85,B 0,C 180,E1 -2032.192,E2 -2032.192} C_VEL
LIN {X 0,Y 573.157,Z 369.094,A -85,B 0,C 180,E1 -2034.808,E2 -2034.808} C_VEL
LIN {X 0,Y 573.116,Z 369.328,A -85,B 0,C 180,E1 -2035.661,E2 -2035.661} C_VEL
LIN {X 0,Y 573.096,Z 372.041,A -85,B 0,C 180,E1 -2038.175,E2 -2038.175} C_VEL
LIN {X 0,Y 573.081,Z 374.682,A -85,B 0,C 180,E1 -2040.624,E2 -2040.624} C_VEL
LIN {X 0,Y 573.063,Z 377.962,A -85,B 0,C 180,E1 -2043.543,E2 -2043.543} C_VEL
LIN {X 0,Y 573.006,Z 380.858,A -85,B 0,C 180,E1 -2046.124,E2 -2046.124} C_VEL
LIN {X 0,Y 572.985,Z 384.65,A -85,B 0,C 180,E1 -2049.163,E2 -2049.163} C_VEL
LIN {X 0,Y 572.945,Z 388.494,A -85,B 0,C 180,E1 -2052.142,E2 -2052.142} C_VEL
LIN {X 0,Y 572.958,Z 391.376,A -85,B 0,C 180,E1 -2054.344,E2 -2054.344} C_VEL
LIN {X 0,Y 572.989,Z 394.259,A -85,B 0,C 180,E1 -2056.524,E2 -2056.524} C_VEL
LIN {X 0,Y 573.011,Z 395.67,A -85,B 0,C 180,E1 -2057.583,E2 -2057.583} C_VEL
LIN {X 0,Y 573.828,Z 402.343,A -85,B 0,C 180,E1 -2057.758,E2 -2057.758} C_VEL
LIN {X 0,Y 573.726,Z 415.763,A -85,B 0,C 180,E1 -2058.16,E2 -2058.16} C_VEL
LIN {X 0,Y 573.629,Z 428.289,A -85,B 0,C 180,E1 -2058.695,E2 -2058.695} C_VEL
LIN {X 0,Y 573.501,Z 439.474,A -85,B 0,C 180,E1 -2059.319,E2 -2059.319} C_VEL
LIN {X 0,Y 573.353,Z 450.833,A -85,B 0,C 180,E1 -2060.119,E2 -2060.119} C_VEL
LIN {X 0,Y 573.28,Z 460.885,A -85,B 0,C 180,E1 -2061.007,E2 -2061.007} C_VEL
LIN {X 0,Y 573.161,Z 470.587,A -85,B 0,C 180,E1 -2062.071,E2 -2062.071} C_VEL
LIN {X 0,Y 573.093,Z 478.523,A -85,B 0,C 180,E1 -2063.163,E2 -2063.163} C_VEL
LIN {X 0,Y 573.07,Z 485.449,A -85,B 0,C 180,E1 -2064.37,E2 -2064.37} C_VEL
LIN {X 0,Y 573.028,Z 490.19,A -85,B 0,C 180,E1 -2065.428,E2 -2065.428} C_VEL
LIN {X 0,Y 573.022,Z 493.823,A -85,B 0,C 180,E1 -2066.484,E2 -2066.484} C_VEL
LIN {X 0,Y 572.959,Z 495.7,A -85,B 0,C 180,E1 -2067.188,E2 -2067.188} C_VEL
LIN {X 0,Y 572.94,Z 497.128,A -85,B 0,C 180,E1 -2067.891,E2 -2067.891} C_VEL
LIN {X 0,Y 572.941,Z 498.755,A -85,B 0,C 180,E1 -2069.297,E2 -2069.297} C_VEL
LIN {X 0,Y 572.939,Z 498.996,A -85,B 0,C 180,E1 -2070,E2 -2070} C_VEL
LIN {X 0,Y 572.94,Z 498.815,A -85,B 0,C 180,E1 -2070.703,E2 -2070.703} C_VEL
LIN {X 0,Y 572.94,Z 497.27,A -85,B 0,C 180,E1 -2072.109,E2 -2072.109} C_VEL
LIN {X 0,Y 572.96,Z 495.909,A -85,B 0,C 180,E1 -2072.812,E2 -2072.812} C_VEL
LIN {X 0,Y 573.015,Z 493.032,A -85,B 0,C 180,E1 -2073.868,E2 -2073.868} C_VEL
LIN {X 0,Y 572.963,Z 489.131,A -85,B 0,C 180,E1 -2074.926,E2 -2074.926} C_VEL
LIN {X 0,Y 573.076,Z 484.098,A -85,B 0,C 180,E1 -2075.984,E2 -2075.984} C_VEL
LIN {X 0,Y 573.083,Z 477.775,A -85,B 0,C 180,E1 -2077.044,E2 -2077.044} C_VEL
LIN {X 0,Y 573.175,Z 469.854,A -85,B 0,C 180,E1 -2078.106,E2 -2078.106} C_VEL
LIN {X 0,Y 573.287,Z 460.004,A -85,B 0,C 180,E1 -2079.17,E2 -2079.17} C_VEL
LIN {X 0,Y 573.423,Z 449.682,A -85,B 0,C 180,E1 -2080.058,E2 -2080.058} C_VEL
LIN {X 0,Y 573.524,Z 438.14,A -85,B 0,C 180,E1 -2080.854,E2 -2080.854} C_VEL
LIN {X 0,Y 573.641,Z 426.516,A -85,B 0,C 180,E1 -2081.482,E2 -2081.482} C_VEL
LIN {X 0,Y 573.723,Z 414.604,A -85,B 0,C 180,E1 -2081.97,E2 -2081.97} C_VEL
LIN {X 0,Y 573.842,Z 401.435,A -85,B 0,C 180,E1 -2082.354,E2 -2082.354} C_VEL
LIN {X 0,Y 572.981,Z 395.67,A -85,B 0,C 180,E1 -2082.508,E2 -2082.508} C_VEL
LIN {X 0,Y 572.958,Z 392.456,A -85,B 0,C 180,E1 -2084.927,E2 -2084.927} C_VEL
LIN {X 0,Y 572.977,Z 389.572,A -85,B 0,C 180,E1 -2087.12,E2 -2087.12} C_VEL
LIN {X 0,Y 572.987,Z 385.727,A -85,B 0,C 180,E1 -2090.087,E2 -2090.087} C_VEL
LIN {X 0,Y 572.991,Z 381.881,A -85,B 0,C 180,E1 -2093.11,E2 -2093.11} C_VEL
LIN {X 0,Y 573.079,Z 378.361,A -85,B 0,C 180,E1 -2096.199,E2 -2096.199} C_VEL
LIN {X 0,Y 573.049,Z 375.685,A -85,B 0,C 180,E1 -2098.575,E2 -2098.575} C_VEL
LIN {X 0,Y 573.111,Z 373.023,A -85,B 0,C 180,E1 -2101.001,E2 -2101.001} C_VEL
LIN {X 0,Y 573.125,Z 370.321,A -85,B 0,C 180,E1 -2103.503,E2 -2103.503} C_VEL
LIN {X 0,Y 573.127,Z 369.098,A -85,B 0,C 180,E1 -2104.755,E2 -2104.755} C_VEL
LIN {X 0,Y 573.256,Z 369.081,A -85,B 0,C 180,E1 -2107.166,E2 -2107.166} C_VEL
LIN {X 0,Y 573.244,Z 369.076,A -85,B 0,C 180,E1 -2109.608,E2 -2109.608} C_VEL
LIN {X 0,Y 573.248,Z 369.078,A -85,B 0,C 180,E1 -2112.642,E2 -2112.642} C_VEL
LIN {X 0,Y 573.219,Z 369.083,A -85,B 0,C 180,E1 -2115.326,E2 -2115.326} C_VEL
LIN {X 0,Y 573.244,Z 369.081,A -85,B 0,C 180,E1 -2117.6,E2 -2117.6} C_VEL
LIN {X 0,Y 573.257,Z 369.079,A -85,B 0,C 180,E1 -2120.567,E2 -2120.567} C_VEL
LIN {X 0,Y 573.257,Z 369.075,A -85,B 0,C 180,E1 -2123.078,E2 -2123.078} C_VEL
LIN {X 0,Y 573.276,Z 369.076,A -85,B 0,C 180,E1 -2125.672,E2 -2125.672} C_VEL
LIN {X 0,Y 573.246,Z 369.077,A -85,B 0,C 180,E1 -2128.185,E2 -2128.185} C_VEL
LIN {X 0,Y 573.268,Z 369.076,A -85,B 0,C 180,E1 -2130.634,E2 -2130.634} C_VEL
LIN {X 0,Y 573.255,Z 369.079,A -85,B 0,C 180,E1 -2133.024,E2 -2133.024} C_VEL
LIN {X 0,Y 573.281,Z 369.072,A -85,B 0,C 180,E1 -2135.366,E2 -2135.366} C_VEL
LIN {X 0,Y 573.234,Z 369.079,A -85,B 0,C 180,E1 -2138.419,E2 -2138.419} C_VEL
LIN {X 0,Y 573.285,Z 369.072,A -85,B 0,C 180,E1 -2140.728,E2 -2140.728} C_VEL
LIN {X 0,Y 573.248,Z 369.077,A -85,B 0,C 180,E1 -2143.622,E2 -2143.622} C_VEL
LIN {X 0,Y 573.279,Z 369.073,A -85,B 0,C 180,E1 -2145.807,E2 -2145.807} C_VEL
LIN {X 0,Y 573.269,Z 369.074,A -85,B 0,C 180,E1 -2148.745,E2 -2148.745} C_VEL
LIN {X 0,Y 573.261,Z 369.081,A -85,B 0,C 180,E1 -2151.54,E2 -2151.54} C_VEL
LIN {X 0,Y 573.246,Z 369.079,A -85,B 0,C 180,E1 -2153.665,E2 -2153.665} C_VEL
LIN {X 0,Y 573.225,Z 369.079,A -85,B 0,C 180,E1 -2155.781,E2 -2155.781} C_VEL
LIN {X 0,Y 573.308,Z 369.07,A -85,B 0,C 180,E1 -2157.892,E2 -2157.892} C_VEL
LIN {X 0,Y 573.336,Z 369.066,A -85,B 0,C 180,E1 -2160.702,E2 -2160.702} C_VEL
LIN {X 0,Y 573.31,Z 369.068,A -85,B 0,C 180,E1 -2162.811,E2 -2162.811} C_VEL
LIN {X 0,Y 573.294,Z 369.073,A -85,B 0,C 180,E1 -2165.628,E2 -2165.628} C_VEL
LIN {X 0,Y 573.294,Z 369.075,A -85,B 0,C 180,E1 -2168.459,E2 -2168.459} C_VEL
LIN {X 0,Y 573.278,Z 369.073,A -85,B 0,C 180,E1 -2171.312,E2 -2171.312} C_VEL
LIN {X 0,Y 573.288,Z 369.071,A -85,B 0,C 180,E1 -2174.424,E2 -2174.424} C_VEL
LIN {X 0,Y 573.263,Z 369.079,A -85,B 0,C 180,E1 -2177.111,E2 -2177.111} C_VEL
LIN {X 0,Y 573.258,Z 369.076,A -85,B 0,C 180,E1 -2180.076,E2 -2180.076} C_VEL
LIN {X 0,Y 573.24,Z 369.077,A -85,B 0,C 180,E1 -2183.099,E2 -2183.099} C_VEL
LIN {X 0,Y 573.259,Z 369.077,A -85,B 0,C 180,E1 -2185.41,E2 -2185.41} C_VEL
LIN {X 0,Y 573.255,Z 369.076,A -85,B 0,C 180,E1 -2188.029,E2 -2188.029} C_VEL
LIN {X 0,Y 573.251,Z 369.075,A -85,B 0,C 180,E1 -2190.176,E2 -2190.176} C_VEL
LIN {X 0,Y 573.258,Z 369.082,A -85,B 0,C 180,E1 -2192.645,E2 -2192.645} C_VEL
LIN {X 0,Y 573.213,Z 369.081,A -85,B 0,C 180,E1 -2195.188,E2 -2195.188} C_VEL
LIN {X 0,Y 573.24,Z 369.083,A -85,B 0,C 180,E1 -2197.807,E2 -2197.807} C_VEL
LIN {X 0,Y 573.249,Z 369.076,A -85,B 0,C 180,E1 -2200.525,E2 -2200.525} C_VEL
LIN {X 0,Y 573.243,Z 369.078,A -85,B 0,C 180,E1 -2203.359,E2 -2203.359} C_VEL
LIN {X 0,Y 573.257,Z 369.082,A -85,B 0,C 180,E1 -2206.33,E2 -2206.33} C_VEL
LIN {X 0,Y 573.248,Z 369.078,A -85,B 0,C 180,E1 -2208.544,E2 -2208.544} C_VEL
LIN {X 0,Y 573.245,Z 369.083,A -85,B 0,C 180,E1 -2211.298,E2 -2211.298} C_VEL
LIN {X 0,Y 573.31,Z 369.282,A -85,B 0,C 180,E1 -2213.301,E2 -2213.301} C_VEL
LIN {X 0,Y 573.798,Z 373.915,A -85,B 0,C 180,E1 -2214.853,E2 -2214.853} C_VEL
LIN {X 0,Y 573.728,Z 381.859,A -85,B 0,C 180,E1 -2217.385,E2 -2217.385} C_VEL
LIN {X 0,Y 573.58,Z 391.8,A -85,B 0,C 180,E1 -2220.454,E2 -2220.454} C_VEL
LIN {X 0,Y 573.497,Z 400.394,A -85,B 0,C 180,E1 -2223.036,E2 -2223.036} C_VEL
LIN {X 0,Y 573.401,Z 409.661,A -85,B 0,C 180,E1 -2225.757,E2 -2225.757} C_VEL
LIN {X 0,Y 573.325,Z 418.928,A -85,B 0,C 180,E1 -2228.423,E2 -2228.423} C_VEL
LIN {X 0,Y 573.221,Z 428.329,A -85,B 0,C 180,E1 -2231.077,E2 -2231.077} C_VEL
LIN {X 0,Y 573.166,Z 438.787,A -85,B 0,C 180,E1 -2233.985,E2 -2233.985} C_VEL
LIN {X 0,Y 573.115,Z 449.378,A -85,B 0,C 180,E1 -2236.887,E2 -2236.887} C_VEL
LIN {X 0,Y 573.113,Z 451.53,A -85,B 0,C 180,E1 -2237.473,E2 -2237.473} C_VEL
LIN {X 0,Y 573.883,Z 458.363,A -85,B 0,C 180,E1 -2237.625,E2 -2237.625} C_VEL
LIN {X 0,Y 573.79,Z 470.491,A -85,B 0,C 180,E1 -2237.937,E2 -2237.937} C_VEL
LIN {X 0,Y 573.684,Z 482.747,A -85,B 0,C 180,E1 -2238.393,E2 -2238.393} C_VEL
LIN {X 0,Y 573.583,Z 494.309,A -85,B 0,C 180,E1 -2238.968,E2 -2238.968} C_VEL
LIN {X 0,Y 573.453,Z 505.476,A -85,B 0,C 180,E1 -2239.674,E2 -2239.674} C_VEL
LIN {X 0,Y 573.308,Z 515.645,A -85,B 0,C 180,E1 -2240.474,E2 -2240.474} C_VEL
LIN {X 0,Y 573.215,Z 524.786,A -85,B 0,C 180,E1 -2241.362,E2 -2241.362} C_VEL
LIN {X 0,Y 573.142,Z 533.69,A -85,B 0,C 180,E1 -2242.425,E2 -2242.425} C_VEL
LIN {X 0,Y 573.051,Z 540.405,A -85,B 0,C 180,E1 -2243.415,E2 -2243.415} C_VEL
LIN {X 0,Y 573.07,Z 545.68,A -85,B 0,C 180,E1 -2244.37,E2 -2244.37} C_VEL
LIN {X 0,Y 573.028,Z 550.371,A -85,B 0,C 180,E1 -2245.427,E2 -2245.427} C_VEL
LIN {X 0,Y 573.022,Z 553.956,A -85,B 0,C 180,E1 -2246.484,E2 -2246.484} C_VEL
LIN {X 0,Y 572.959,Z 555.808,A -85,B 0,C 180,E1 -2247.188,E2 -2247.188} C_VEL
LIN {X 0,Y 572.939,Z 557.201,A -85,B 0,C 180,E1 -2247.891,E2 -2247.891} C_VEL
LIN {X 0,Y 572.941,Z 558.784,A -85,B 0,C 180,E1 -2249.297,E2 -2249.297} C_VEL
LIN {X 0,Y 572.938,Z 559,A -85,B 0,C 180,E1 -2250,E2 -2250} C_VEL
LIN {X 0,Y 572.946,Z 558.185,A -85,B 0,C 180,E1 -2251.406,E2 -2251.406} C_VEL
LIN {X 0,Y 572.94,Z 557.201,A -85,B 0,C 180,E1 -2252.109,E2 -2252.109} C_VEL
LIN {X 0,Y 572.959,Z 555.81,A -85,B 0,C 180,E1 -2252.812,E2 -2252.812} C_VEL
LIN {X 0,Y 573.014,Z 552.896,A -85,B 0,C 180,E1 -2253.868,E2 -2253.868} C_VEL
LIN {X 0,Y 572.963,Z 548.95,A -85,B 0,C 180,E1 -2254.926,E2 -2254.926} C_VEL
LIN {X 0,Y 573.064,Z 542.878,A -85,B 0,C 180,E1 -2256.16,E2 -2256.16} C_VEL
LIN {X 0,Y 573.119,Z 536.236,A -85,B 0,C 180,E1 -2257.221,E2 -2257.221} C_VEL
LIN {X 0,Y 573.201,Z 527.99,A -85,B 0,C 180,E1 -2258.283,E2 -2258.283} C_VEL
LIN {X 0,Y 573.287,Z 519.537,A -85,B 0,C 180,E1 -2259.17,E2 -2259.17} C_VEL
LIN {X 0,Y 573.429,Z 509.094,A -85,B 0,C 180,E1 -2260.058,E2 -2260.058} C_VEL
LIN {X 0,Y 573.507,Z 498.828,A -85,B 0,C 180,E1 -2260.766,E2 -2260.766} C_VEL
LIN {X 0,Y 573.628,Z 487.591,A -85,B 0,C 180,E1 -2261.385,E2 -2261.385} C_VEL
LIN {X 0,Y 573.709,Z 475.767,A -85,B 0,C 180,E1 -2261.885,E2 -2261.885} C_VEL
LIN {X 0,Y 573.841,Z 462.35,A -85,B 0,C 180,E1 -2262.286,E2 -2262.286} C_VEL
LIN {X 0,Y 573.696,Z 455.373,A -85,B 0,C 180,E1 -2262.438,E2 -2262.438} C_VEL
LIN {X 0,Y 573.113,Z 451.53,A -85,B 0,C 180,E1 -2262.527,E2 -2262.527} C_VEL
LIN {X 0,Y 573.164,Z 441.435,A -85,B 0,C 180,E1 -2265.285,E2 -2265.285} C_VEL
LIN {X 0,Y 573.215,Z 430.844,A -85,B 0,C 180,E1 -2268.219,E2 -2268.219} C_VEL
LIN {X 0,Y 573.31,Z 421.577,A -85,B 0,C 180,E1 -2270.824,E2 -2270.824} C_VEL
LIN {X 0,Y 573.371,Z 412.311,A -85,B 0,C 180,E1 -2273.476,E2 -2273.476} C_VEL
LIN {X 0,Y 573.459,Z 404.366,A -85,B 0,C 180,E1 -2275.79,E2 -2275.79} C_VEL
LIN {X 0,Y 573.558,Z 395.099,A -85,B 0,C 180,E1 -2278.547,E2 -2278.547} C_VEL
LIN {X 0,Y 573.659,Z 385.831,A -85,B 0,C 180,E1 -2281.378,E2 -2281.378} C_VEL
LIN {X 0,Y 573.786,Z 377.778,A -85,B 0,C 180,E1 -2283.905,E2 -2283.905} C_VEL
LIN {X 0,Y 573.751,Z 372.592,A -85,B 0,C 180,E1 -2285.58,E2 -2285.58} C_VEL
LIN {X 0,Y 573.264,Z 369.081,A -85,B 0,C 180,E1 -2286.812,E2 -2286.812} C_VEL
LIN {X 0,Y 573.241,Z 369.079,A -85,B 0,C 180,E1 -2289.608,E2 -2289.608} C_VEL
LIN {X 0,Y 573.247,Z 369.078,A -85,B 0,C 180,E1 -2292.642,E2 -2292.642} C_VEL
LIN {X 0,Y 573.226,Z 369.087,A -85,B 0,C 180,E1 -2295.325,E2 -2295.325} C_VEL
LIN {X 0,Y 573.243,Z 369.078,A -85,B 0,C 180,E1 -2297.6,E2 -2297.6} C_VEL
LIN {X 0,Y 573.251,Z 369.08,A -85,B 0,C 180,E1 -2300.393,E2 -2300.393} C_VEL
LIN {X 0,Y 573.256,Z 369.075,A -85,B 0,C 180,E1 -2303.078,E2 -2303.078} C_VEL
LIN {X 0,Y 573.272,Z 369.079,A -85,B 0,C 180,E1 -2305.672,E2 -2305.672} C_VEL
LIN {X 0,Y 573.245,Z 369.076,A -85,B 0,C 180,E1 -2308.185,E2 -2308.185} C_VEL
LIN {X 0,Y 573.268,Z 369.078,A -85,B 0,C 180,E1 -2310.634,E2 -2310.634} C_VEL
LIN {X 0,Y 573.255,Z 369.076,A -85,B 0,C 180,E1 -2313.024,E2 -2313.024} C_VEL
LIN {X 0,Y 573.279,Z 369.073,A -85,B 0,C 180,E1 -2315.366,E2 -2315.366} C_VEL
LIN {X 0,Y 573.233,Z 369.078,A -85,B 0,C 180,E1 -2318.419,E2 -2318.419} C_VEL
LIN {X 0,Y 573.283,Z 369.074,A -85,B 0,C 180,E1 -2320.728,E2 -2320.728} C_VEL
